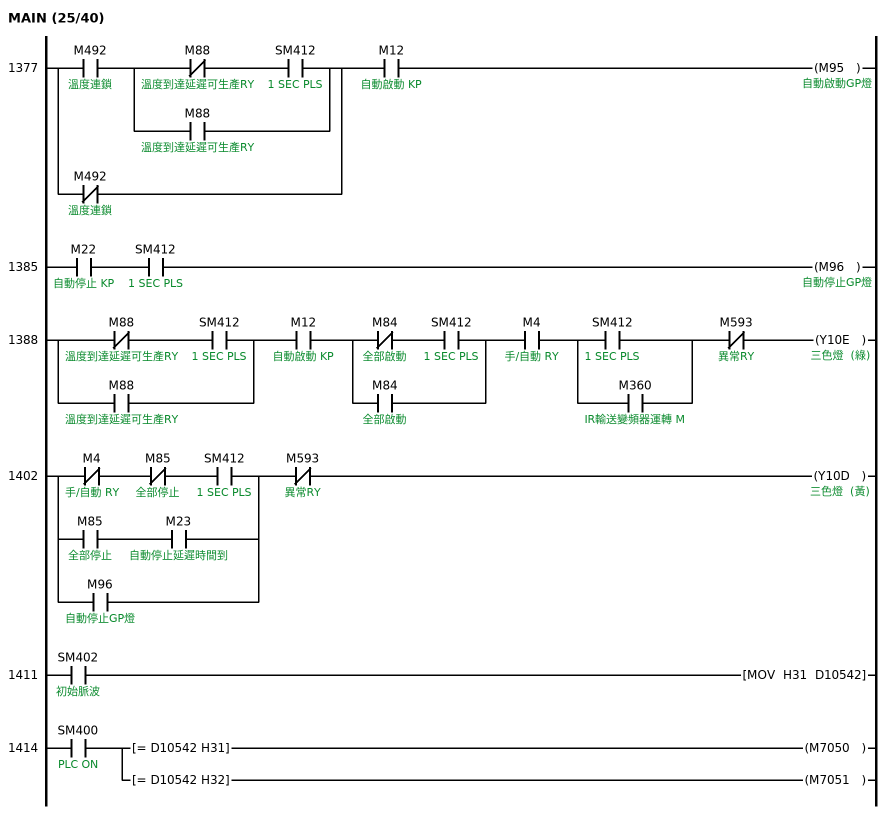
[picture p24: ladder of MAIN, rungs at steps 1377 to 1414]
1377  LD      M492  ; 溫度連鎖
      LDI     M88  ; 溫度到達延遲可生產RY
      AND     SM412  ; 1 SEC PLS
      OR      M88  ; 溫度到達延遲可生產RY
      ANB
      ORI     M492  ; 溫度連鎖
      AND     M12  ; 自動啟動 KP
      OUT     M95  ; 自動啟動GP燈
1385  LD      M22  ; 自動停止 KP
      AND     SM412  ; 1 SEC PLS
      OUT     M96  ; 自動停止GP燈
1388  LDI     M88  ; 溫度到達延遲可生產RY
      AND     SM412  ; 1 SEC PLS
      OR      M88  ; 溫度到達延遲可生產RY
      AND     M12  ; 自動啟動 KP
      LDI     M84  ; 全部啟動
      AND     SM412  ; 1 SEC PLS
      OR      M84  ; 全部啟動
      ANB
      AND     M4  ; 手/自動 RY
      LD      SM412  ; 1 SEC PLS
      OR      M360  ; IR輸送變頻器運轉 M
      ANB
      ANI     M593  ; 異常RY
      OUT     Y10E  ; 三色燈  (綠)
1402  LDI     M4  ; 手/自動 RY
      ANI     M85  ; 全部停止
      AND     SM412  ; 1 SEC PLS
      LD      M85  ; 全部停止
      AND     M23  ; 自動停止延遲時間到
      ORB
      OR      M96  ; 自動停止GP燈
      ANI     M593  ; 異常RY
      OUT     Y10D  ; 三色燈  (黃)
1411  LD      SM402  ; 初始脈波
      MOV     H31 D10542
1414  LD      SM400  ; PLC ON
      MPS
      AND=    D10542 H31
      OUT     M7050
      MPP
      AND=    D10542 H32
      OUT     M7051
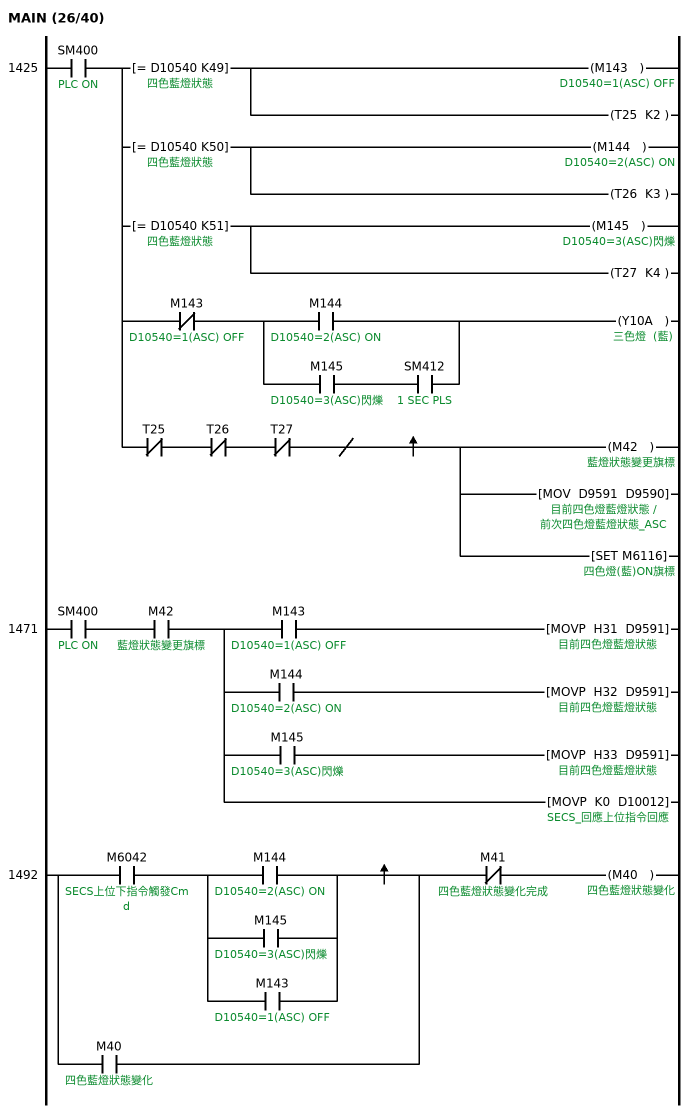
1425  LD      SM400  ; PLC ON
      MPS
      AND=    D10540 K49  ; 四色藍燈狀態
      OUT     M143  ; D10540=1(ASC) OFF
      OUT     T25 K2
      MRD
      AND=    D10540 K50  ; 四色藍燈狀態
      OUT     M144  ; D10540=2(ASC) ON
      OUT     T26 K3
      MRD
      AND=    D10540 K51  ; 四色藍燈狀態
      OUT     M145  ; D10540=3(ASC)閃爍
      OUT     T27 K4
      MRD
      ANI     M143  ; D10540=1(ASC) OFF
      LD      M144  ; D10540=2(ASC) ON
      LD      M145  ; D10540=3(ASC)閃爍
      AND     SM412  ; 1 SEC PLS
      ORB
      ANB
      OUT     Y10A  ; 三色燈  (藍)
      MPP
      ANI     T25
      ANI     T26
      ANI     T27
      INV
      MEP
      OUT     M42  ; 藍燈狀態變更旗標
      MOV     D9591 D9590  ; 目前四色燈藍燈狀態 / 前次四色燈藍燈狀態_ASC
      SET     M6116  ; 四色燈(藍)ON旗標
1471  LD      SM400  ; PLC ON
      AND     M42  ; 藍燈狀態變更旗標
      MPS
      AND     M143  ; D10540=1(ASC) OFF
      MOVP    H31 D9591
      MRD
      AND     M144  ; D10540=2(ASC) ON
      MOVP    H32 D9591
      MRD
      AND     M145  ; D10540=3(ASC)閃爍
      MOVP    H33 D9591
      MPP
      MOVP    K0 D10012  ; SECS_回應上位指令回應
1492  LD      M6042  ; SECS上位下指令觸發Cmd
      LD      M144  ; D10540=2(ASC) ON
      OR      M145  ; D10540=3(ASC)閃爍
      OR      M143  ; D10540=1(ASC) OFF
      ANB
      MEP
      OR      M40  ; 四色藍燈狀態變化
      ANI     M41  ; 四色藍燈狀態變化完成
      OUT     M40  ; 四色藍燈狀態變化
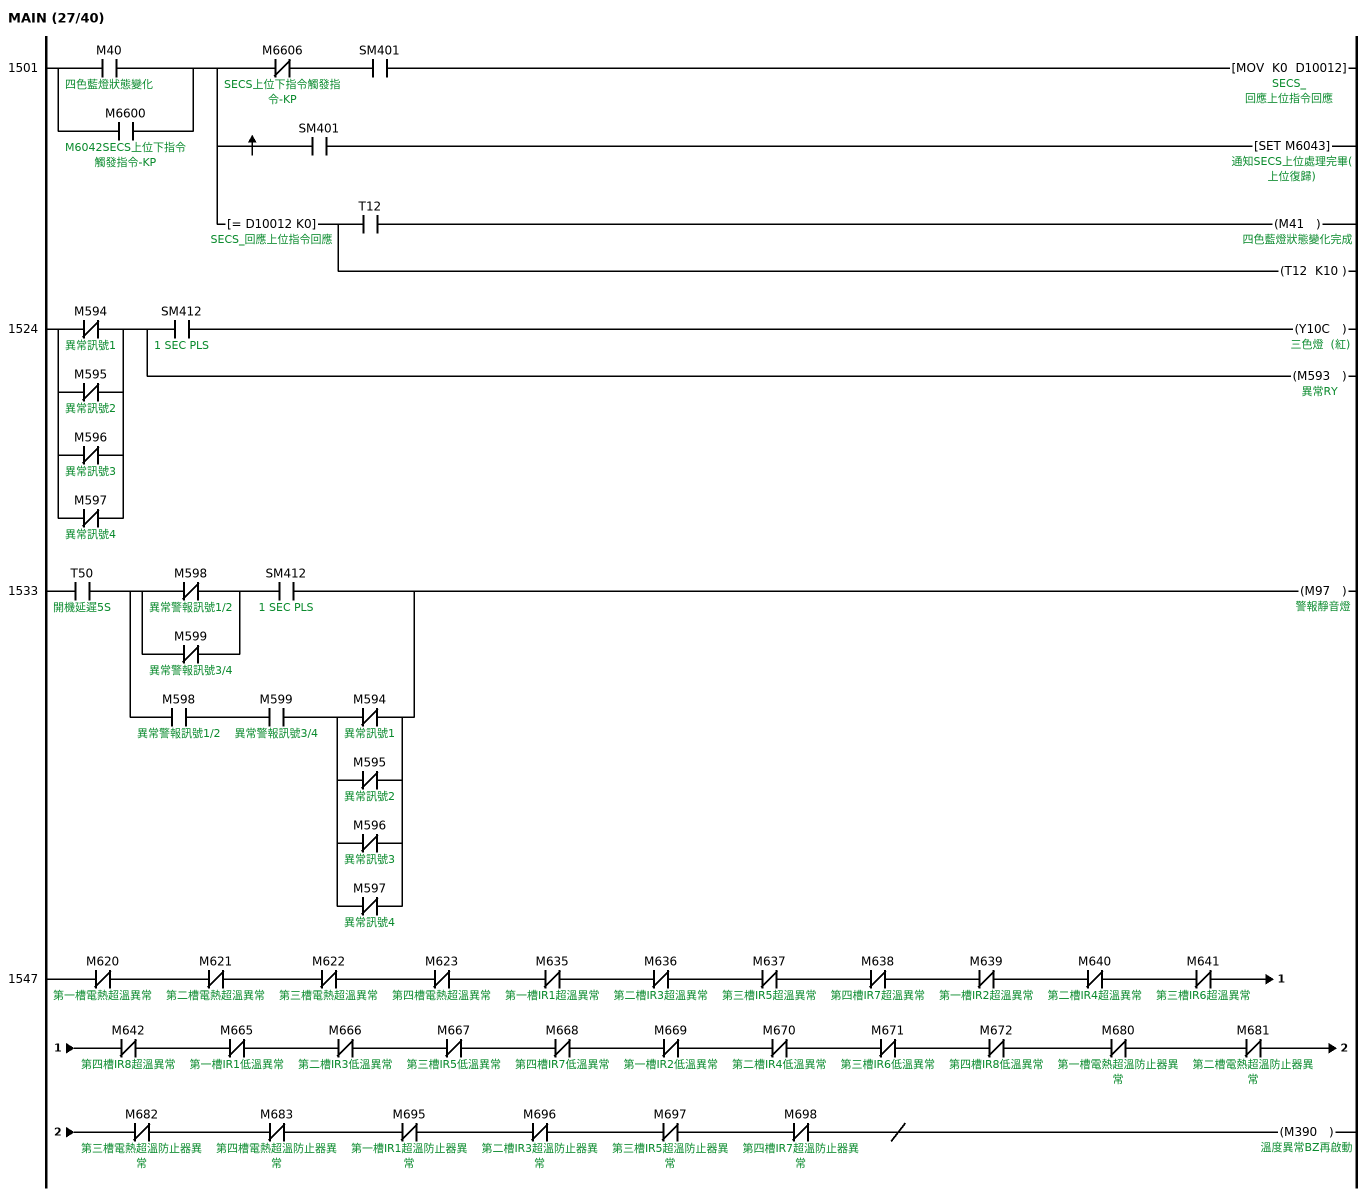
1501  LD      M40  ; 四色藍燈狀態變化
      OR      M6600  ; M6042SECS上位下指令觸發指令-KP
      MPS
      ANI     M6606  ; SECS上位下指令觸發指令-KP
      AND     SM401
      MOV     K0 D10012
      MRD
      MEP
      AND     SM401
      SET     M6043  ; 通知SECS上位處理完畢(上位復歸)
      MPP
      AND=    D10012 K0  ; SECS_回應上位指令回應
      MPS
      AND     T12
      OUT     M41  ; 四色藍燈狀態變化完成
      MPP
      OUT     T12 K10
1524  LDI     M594  ; 異常訊號1
      ORI     M595  ; 異常訊號2
      ORI     M596  ; 異常訊號3
      ORI     M597  ; 異常訊號4
      MPS
      AND     SM412  ; 1 SEC PLS
      OUT     Y10C  ; 三色燈  (紅)
      MPP
      OUT     M593  ; 異常RY
1533  LD      T50  ; 開機延遲5S
      LDI     M598  ; 異常警報訊號1/2
      ORI     M599  ; 異常警報訊號3/4
      AND     SM412  ; 1 SEC PLS
      LD      M598  ; 異常警報訊號1/2
      AND     M599  ; 異常警報訊號3/4
      LDI     M594  ; 異常訊號1
      ORI     M595  ; 異常訊號2
      ORI     M596  ; 異常訊號3
      ORI     M597  ; 異常訊號4
      ANB
      ORB
      ANB
      OUT     M97  ; 警報靜音燈
1547  LDI     M620  ; 第一槽電熱超溫異常
      ANI     M621  ; 第二槽電熱超溫異常
      ANI     M622  ; 第三槽電熱超溫異常
      ANI     M623  ; 第四槽電熱超溫異常
      ANI     M635  ; 第一槽IR1超溫異常
      ANI     M636  ; 第二槽IR3超溫異常
      ANI     M637  ; 第三槽IR5超溫異常
      ANI     M638  ; 第四槽IR7超溫異常
      ANI     M639  ; 第一槽IR2超溫異常
      ANI     M640  ; 第二槽IR4超溫異常
      ANI     M641  ; 第三槽IR6超溫異常
      ANI     M642  ; 第四槽IR8超溫異常
      ANI     M665  ; 第一槽IR1低溫異常
      ANI     M666  ; 第二槽IR3低溫異常
      ANI     M667  ; 第三槽IR5低溫異常
      ANI     M668  ; 第四槽IR7低溫異常
      ANI     M669  ; 第一槽IR2低溫異常
      ANI     M670  ; 第二槽IR4低溫異常
      ANI     M671  ; 第三槽IR6低溫異常
      ANI     M672  ; 第四槽IR8低溫異常
      ANI     M680  ; 第一槽電熱超溫防止器異常
      ANI     M681  ; 第二槽電熱超溫防止器異常
      ANI     M682  ; 第三槽電熱超溫防止器異常
      ANI     M683  ; 第四槽電熱超溫防止器異常
      ANI     M695  ; 第一槽IR1超溫防止器異常
      ANI     M696  ; 第二槽IR3超溫防止器異常
      ANI     M697  ; 第三槽IR5超溫防止器異常
      ANI     M698  ; 第四槽IR7超溫防止器異常
      INV
      OUT     M390  ; 溫度異常BZ再啟動
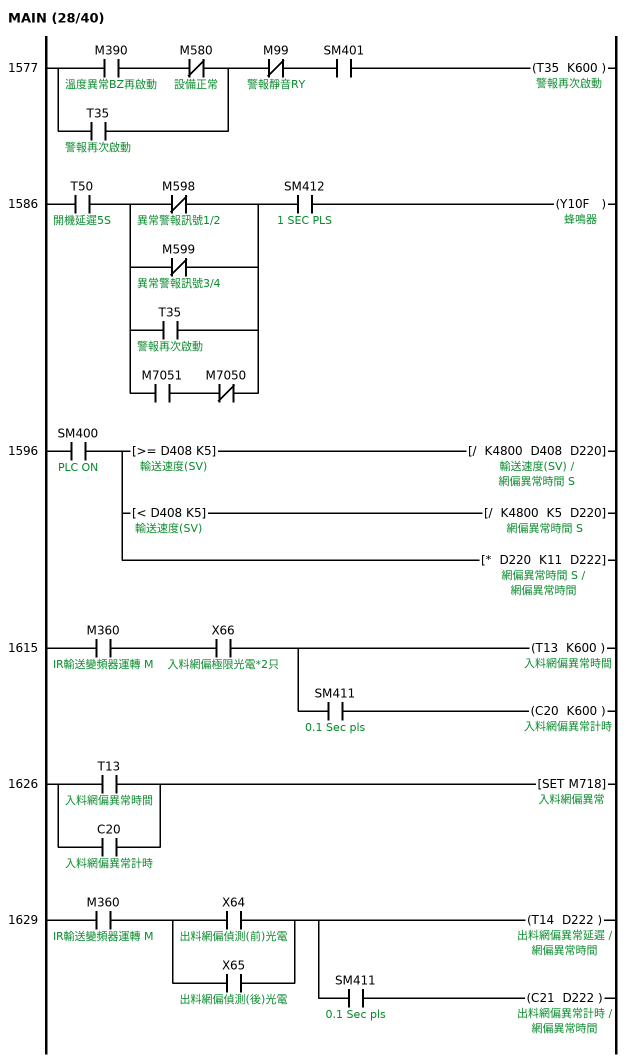
1577  LD      M390  ; 溫度異常BZ再啟動
      ANI     M580  ; 設備正常
      OR      T35  ; 警報再次啟動
      ANI     M99  ; 警報靜音RY
      AND     SM401
      OUT     T35 K600  ; 警報再次啟動
1586  LD      T50  ; 開機延遲5S
      LDI     M598  ; 異常警報訊號1/2
      ORI     M599  ; 異常警報訊號3/4
      OR      T35  ; 警報再次啟動
      LD      M7051
      ANI     M7050
      ORB
      ANB
      AND     SM412  ; 1 SEC PLS
      OUT     Y10F  ; 蜂鳴器
1596  LD      SM400  ; PLC ON
      MPS
      AND>=   D408 K5  ; 輸送速度(SV)
      /       K4800 D408 D220  ; 網偏異常時間 S
      MRD
      AND<    D408 K5  ; 輸送速度(SV)
      /       K4800 K5 D220
      MPP
      *       D220 K11 D222  ; 網偏異常時間
1615  LD      M360  ; IR輸送變頻器運轉 M
      AND     X66  ; 入料網偏極限光電*2只
      OUT     T13 K600  ; 入料網偏異常時間
      AND     SM411  ; 0.1 Sec pls
      OUT     C20 K600  ; 入料網偏異常計時
1626  LD      T13  ; 入料網偏異常時間
      OR      C20  ; 入料網偏異常計時
      SET     M718  ; 入料網偏異常
1629  LD      M360  ; IR輸送變頻器運轉 M
      LD      X64  ; 出料網偏偵測(前)光電
      OR      X65  ; 出料網偏偵測(後)光電
      ANB
      OUT     T14 D222  ; 出料網偏異常延遲 / 網偏異常時間
      AND     SM411  ; 0.1 Sec pls
      OUT     C21 D222  ; 出料網偏異常計時 / 網偏異常時間
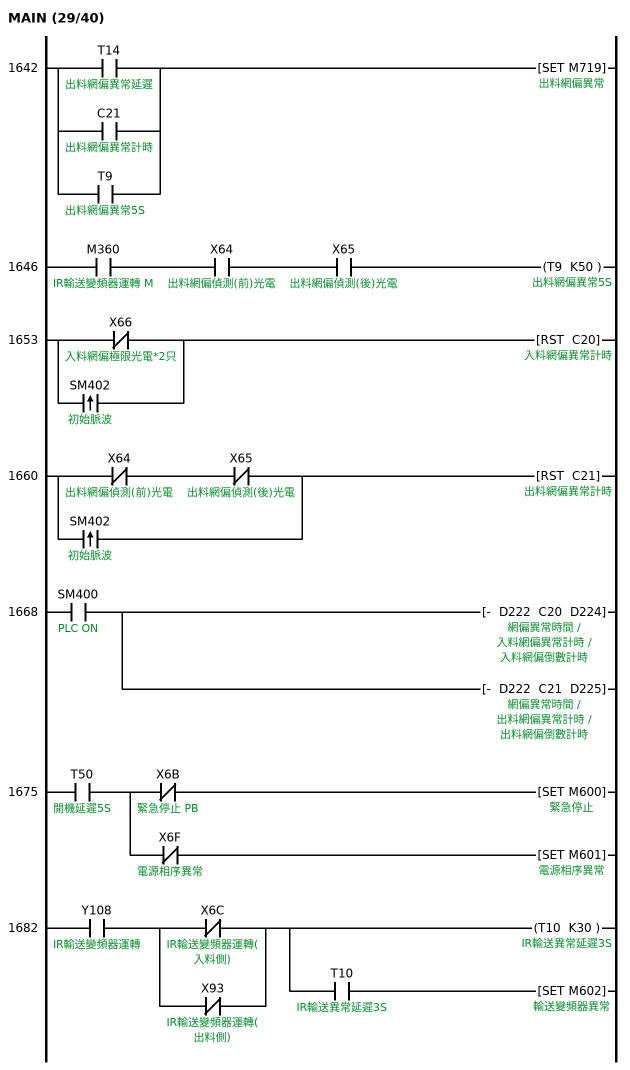
1642  LD      T14  ; 出料網偏異常延遲
      OR      C21  ; 出料網偏異常計時
      OR      T9  ; 出料網偏異常5S
      SET     M719  ; 出料網偏異常
1646  LD      M360  ; IR輸送變頻器運轉 M
      AND     X64  ; 出料網偏偵測(前)光電
      AND     X65  ; 出料網偏偵測(後)光電
      OUT     T9 K50  ; 出料網偏異常5S
1653  LDI     X66  ; 入料網偏極限光電*2只
      ORP     SM402  ; 初始脈波
      RST     C20  ; 入料網偏異常計時
1660  LDI     X64  ; 出料網偏偵測(前)光電
      ANI     X65  ; 出料網偏偵測(後)光電
      ORP     SM402  ; 初始脈波
      RST     C21  ; 出料網偏異常計時
1668  LD      SM400  ; PLC ON
      -       D222 C20 D224  ; 入料網偏倒數計時
      -       D222 C21 D225  ; 出料網偏倒數計時
1675  LD      T50  ; 開機延遲5S
      MPS
      ANI     X6B  ; 緊急停止 PB
      SET     M600  ; 緊急停止
      MPP
      ANI     X6F  ; 電源相序異常
      SET     M601  ; 電源相序異常
1682  LD      Y108  ; IR輸送變頻器運轉
      LDI     X6C  ; IR輸送變頻器運轉(入料側)
      ORI     X93  ; IR輸送變頻器運轉(出料側)
      ANB
      OUT     T10 K30  ; IR輸送異常延遲3S
      AND     T10  ; IR輸送異常延遲3S
      SET     M602  ; 輸送變頻器異常
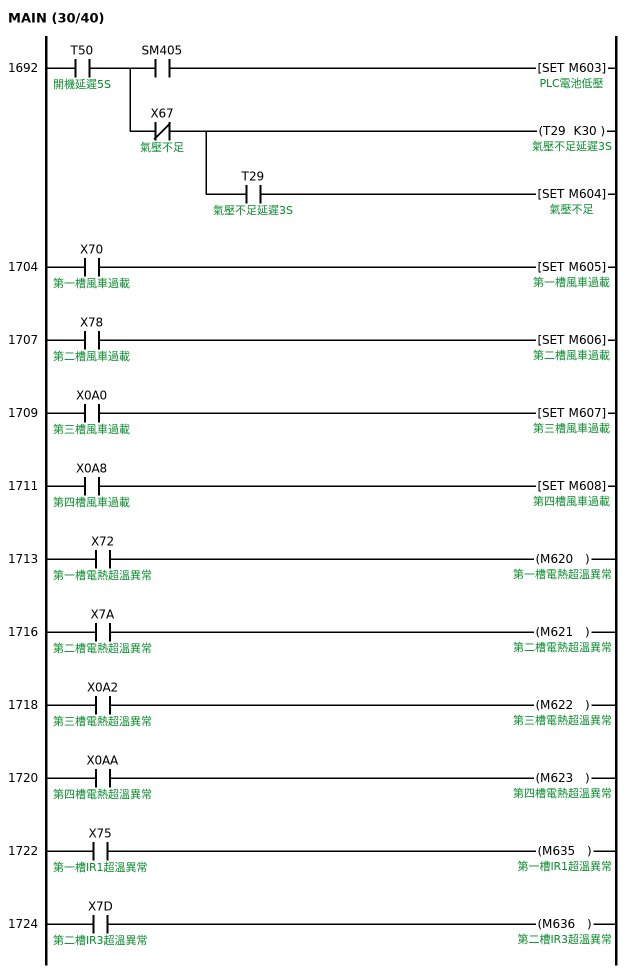
1692  LD      T50  ; 開機延遲5S
      MPS
      AND     SM405
      SET     M603  ; PLC電池低壓
      MPP
      ANI     X67  ; 氣壓不足
      OUT     T29 K30  ; 氣壓不足延遲3S
      AND     T29  ; 氣壓不足延遲3S
      SET     M604  ; 氣壓不足
1704  LD      X70  ; 第一槽風車過載
      SET     M605  ; 第一槽風車過載
        [note] 
1707  LD      X78  ; 第二槽風車過載
      SET     M606  ; 第二槽風車過載
1709  LD      X0A0  ; 第三槽風車過載
      SET     M607  ; 第三槽風車過載
1711  LD      X0A8  ; 第四槽風車過載
      SET     M608  ; 第四槽風車過載
1713  LD      X72  ; 第一槽電熱超溫異常
      OUT     M620  ; 第一槽電熱超溫異常
        [note] 
1716  LD      X7A  ; 第二槽電熱超溫異常
      OUT     M621  ; 第二槽電熱超溫異常
1718  LD      X0A2  ; 第三槽電熱超溫異常
      OUT     M622  ; 第三槽電熱超溫異常
1720  LD      X0AA  ; 第四槽電熱超溫異常
      OUT     M623  ; 第四槽電熱超溫異常
1722  LD      X75  ; 第一槽IR1超溫異常
      OUT     M635  ; 第一槽IR1超溫異常
1724  LD      X7D  ; 第二槽IR3超溫異常
      OUT     M636  ; 第二槽IR3超溫異常
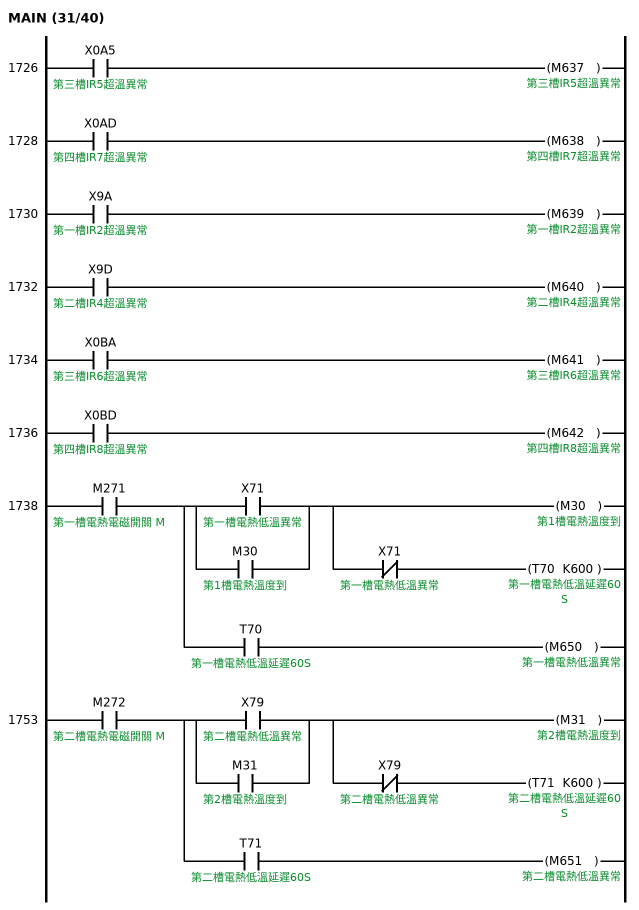
1726  LD      X0A5  ; 第三槽IR5超溫異常
      OUT     M637  ; 第三槽IR5超溫異常
1728  LD      X0AD  ; 第四槽IR7超溫異常
      OUT     M638  ; 第四槽IR7超溫異常
1730  LD      X9A  ; 第一槽IR2超溫異常
      OUT     M639  ; 第一槽IR2超溫異常
1732  LD      X9D  ; 第二槽IR4超溫異常
      OUT     M640  ; 第二槽IR4超溫異常
1734  LD      X0BA  ; 第三槽IR6超溫異常
      OUT     M641  ; 第三槽IR6超溫異常
1736  LD      X0BD  ; 第四槽IR8超溫異常
      OUT     M642  ; 第四槽IR8超溫異常
1738  LD      M271  ; 第一槽電熱電磁開關 M
      MPS
      LD      X71  ; 第一槽電熱低溫異常
      OR      M30  ; 第1槽電熱溫度到
      ANB
      OUT     M30  ; 第1槽電熱溫度到
        [note] 
      ANI     X71  ; 第一槽電熱低溫異常
      OUT     T70 K600  ; 第一槽電熱低溫延遲60S
      MPP
      AND     T70  ; 第一槽電熱低溫延遲60S
      OUT     M650  ; 第一槽電熱低溫異常
1753  LD      M272  ; 第二槽電熱電磁開關 M
      MPS
      LD      X79  ; 第二槽電熱低溫異常
      OR      M31  ; 第2槽電熱溫度到
      ANB
      OUT     M31  ; 第2槽電熱溫度到
      ANI     X79  ; 第二槽電熱低溫異常
      OUT     T71 K600  ; 第二槽電熱低溫延遲60S
      MPP
      AND     T71  ; 第二槽電熱低溫延遲60S
      OUT     M651  ; 第二槽電熱低溫異常
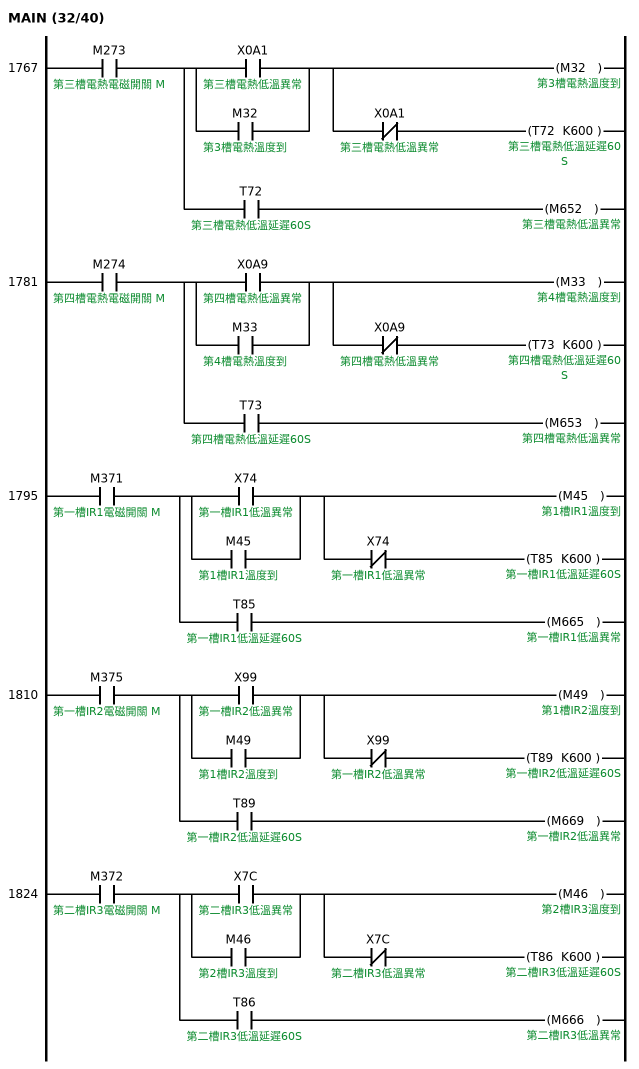
1767  LD      M273  ; 第三槽電熱電磁開關 M
      MPS
      LD      X0A1  ; 第三槽電熱低溫異常
      OR      M32  ; 第3槽電熱溫度到
      ANB
      OUT     M32  ; 第3槽電熱溫度到
      ANI     X0A1  ; 第三槽電熱低溫異常
      OUT     T72 K600  ; 第三槽電熱低溫延遲60S
      MPP
      AND     T72  ; 第三槽電熱低溫延遲60S
      OUT     M652  ; 第三槽電熱低溫異常
1781  LD      M274  ; 第四槽電熱電磁開關 M
      MPS
      LD      X0A9  ; 第四槽電熱低溫異常
      OR      M33  ; 第4槽電熱溫度到
      ANB
      OUT     M33  ; 第4槽電熱溫度到
      ANI     X0A9  ; 第四槽電熱低溫異常
      OUT     T73 K600  ; 第四槽電熱低溫延遲60S
      MPP
      AND     T73  ; 第四槽電熱低溫延遲60S
      OUT     M653  ; 第四槽電熱低溫異常
1795  LD      M371  ; 第一槽IR1電磁開關 M
      MPS
      LD      X74  ; 第一槽IR1低溫異常
      OR      M45  ; 第1槽IR1溫度到
      ANB
      OUT     M45  ; 第1槽IR1溫度到
        [note] 
      ANI     X74  ; 第一槽IR1低溫異常
      OUT     T85 K600  ; 第一槽IR1低溫延遲60S
      MPP
      AND     T85  ; 第一槽IR1低溫延遲60S
      OUT     M665  ; 第一槽IR1低溫異常
1810  LD      M375  ; 第一槽IR2電磁開關 M
      MPS
      LD      X99  ; 第一槽IR2低溫異常
      OR      M49  ; 第1槽IR2溫度到
      ANB
      OUT     M49  ; 第1槽IR2溫度到
      ANI     X99  ; 第一槽IR2低溫異常
      OUT     T89 K600  ; 第一槽IR2低溫延遲60S
      MPP
      AND     T89  ; 第一槽IR2低溫延遲60S
      OUT     M669  ; 第一槽IR2低溫異常
1824  LD      M372  ; 第二槽IR3電磁開關 M
      MPS
      LD      X7C  ; 第二槽IR3低溫異常
      OR      M46  ; 第2槽IR3溫度到
      ANB
      OUT     M46  ; 第2槽IR3溫度到
      ANI     X7C  ; 第二槽IR3低溫異常
      OUT     T86 K600  ; 第二槽IR3低溫延遲60S
      MPP
      AND     T86  ; 第二槽IR3低溫延遲60S
      OUT     M666  ; 第二槽IR3低溫異常
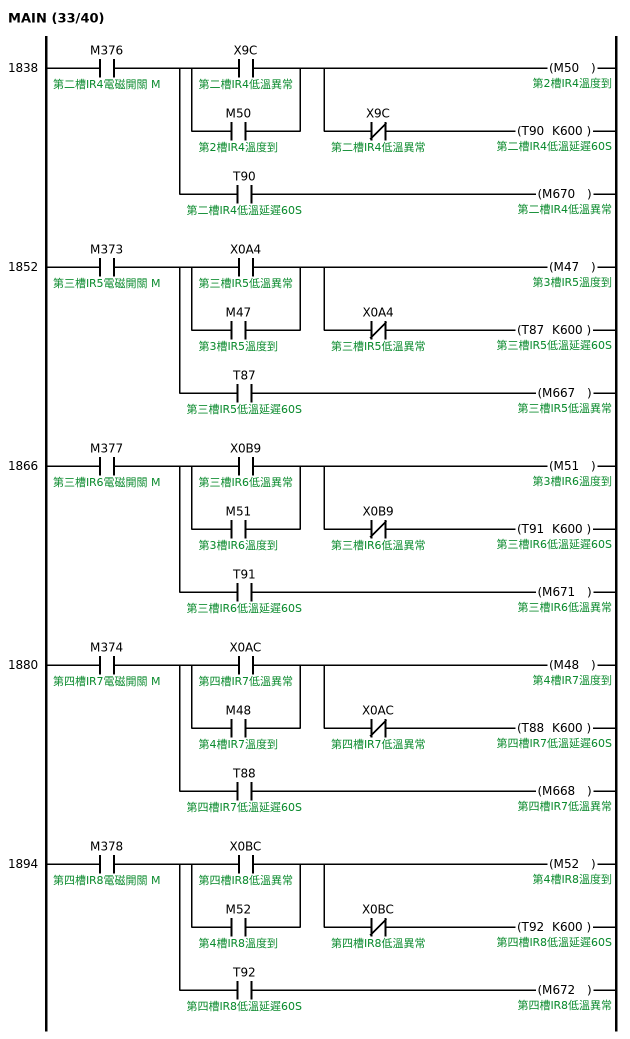
1838  LD      M376  ; 第二槽IR4電磁開關 M
      MPS
      LD      X9C  ; 第二槽IR4低溫異常
      OR      M50  ; 第2槽IR4溫度到
      ANB
      OUT     M50  ; 第2槽IR4溫度到
      ANI     X9C  ; 第二槽IR4低溫異常
      OUT     T90 K600  ; 第二槽IR4低溫延遲60S
      MPP
      AND     T90  ; 第二槽IR4低溫延遲60S
      OUT     M670  ; 第二槽IR4低溫異常
1852  LD      M373  ; 第三槽IR5電磁開關 M
      MPS
      LD      X0A4  ; 第三槽IR5低溫異常
      OR      M47  ; 第3槽IR5溫度到
      ANB
      OUT     M47  ; 第3槽IR5溫度到
      ANI     X0A4  ; 第三槽IR5低溫異常
      OUT     T87 K600  ; 第三槽IR5低溫延遲60S
      MPP
      AND     T87  ; 第三槽IR5低溫延遲60S
      OUT     M667  ; 第三槽IR5低溫異常
1866  LD      M377  ; 第三槽IR6電磁開關 M
      MPS
      LD      X0B9  ; 第三槽IR6低溫異常
      OR      M51  ; 第3槽IR6溫度到
      ANB
      OUT     M51  ; 第3槽IR6溫度到
      ANI     X0B9  ; 第三槽IR6低溫異常
      OUT     T91 K600  ; 第三槽IR6低溫延遲60S
      MPP
      AND     T91  ; 第三槽IR6低溫延遲60S
      OUT     M671  ; 第三槽IR6低溫異常
1880  LD      M374  ; 第四槽IR7電磁開關 M
      MPS
      LD      X0AC  ; 第四槽IR7低溫異常
      OR      M48  ; 第4槽IR7溫度到
      ANB
      OUT     M48  ; 第4槽IR7溫度到
      ANI     X0AC  ; 第四槽IR7低溫異常
      OUT     T88 K600  ; 第四槽IR7低溫延遲60S
      MPP
      AND     T88  ; 第四槽IR7低溫延遲60S
      OUT     M668  ; 第四槽IR7低溫異常
1894  LD      M378  ; 第四槽IR8電磁開關 M
      MPS
      LD      X0BC  ; 第四槽IR8低溫異常
      OR      M52  ; 第4槽IR8溫度到
      ANB
      OUT     M52  ; 第4槽IR8溫度到
      ANI     X0BC  ; 第四槽IR8低溫異常
      OUT     T92 K600  ; 第四槽IR8低溫延遲60S
      MPP
      AND     T92  ; 第四槽IR8低溫延遲60S
      OUT     M672  ; 第四槽IR8低溫異常
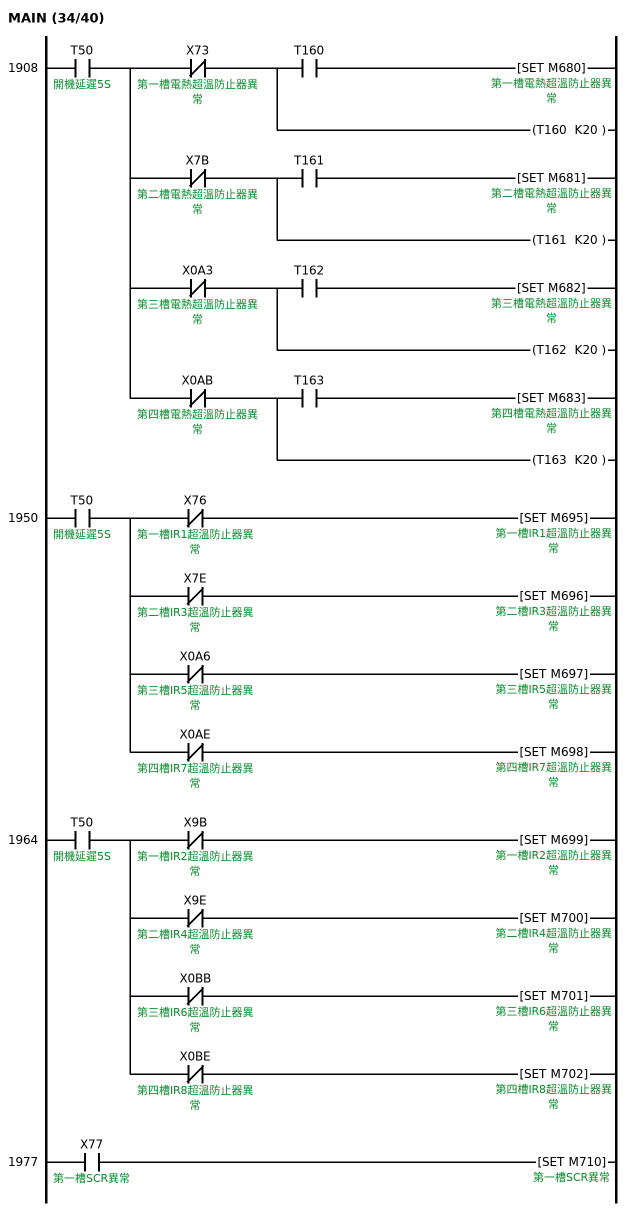
1908  LD      T50  ; 開機延遲5S
      MPS
      ANI     X73  ; 第一槽電熱超溫防止器異常
      MPS
      AND     T160
      SET     M680  ; 第一槽電熱超溫防止器異常
        [note] 
      MPP
      OUT     T160 K20
      MRD
      ANI     X7B  ; 第二槽電熱超溫防止器異常
      MPS
      AND     T161
      SET     M681  ; 第二槽電熱超溫防止器異常
      MPP
      OUT     T161 K20
      MRD
      ANI     X0A3  ; 第三槽電熱超溫防止器異常
      MPS
      AND     T162
      SET     M682  ; 第三槽電熱超溫防止器異常
      MPP
      OUT     T162 K20
      MPP
      ANI     X0AB  ; 第四槽電熱超溫防止器異常
      MPS
      AND     T163
      SET     M683  ; 第四槽電熱超溫防止器異常
      MPP
      OUT     T163 K20
1950  LD      T50  ; 開機延遲5S
      MPS
      ANI     X76  ; 第一槽IR1超溫防止器異常
      SET     M695  ; 第一槽IR1超溫防止器異常
        [note] 
      MRD
      ANI     X7E  ; 第二槽IR3超溫防止器異常
      SET     M696  ; 第二槽IR3超溫防止器異常
      MRD
      ANI     X0A6  ; 第三槽IR5超溫防止器異常
      SET     M697  ; 第三槽IR5超溫防止器異常
      MPP
      ANI     X0AE  ; 第四槽IR7超溫防止器異常
      SET     M698  ; 第四槽IR7超溫防止器異常
1964  LD      T50  ; 開機延遲5S
      MPS
      ANI     X9B  ; 第一槽IR2超溫防止器異常
      SET     M699  ; 第一槽IR2超溫防止器異常
      MRD
      ANI     X9E  ; 第二槽IR4超溫防止器異常
      SET     M700  ; 第二槽IR4超溫防止器異常
      MRD
      ANI     X0BB  ; 第三槽IR6超溫防止器異常
      SET     M701  ; 第三槽IR6超溫防止器異常
      MPP
      ANI     X0BE  ; 第四槽IR8超溫防止器異常
      SET     M702  ; 第四槽IR8超溫防止器異常
1977  LD      X77  ; 第一槽SCR異常
      SET     M710  ; 第一槽SCR異常
        [note] 
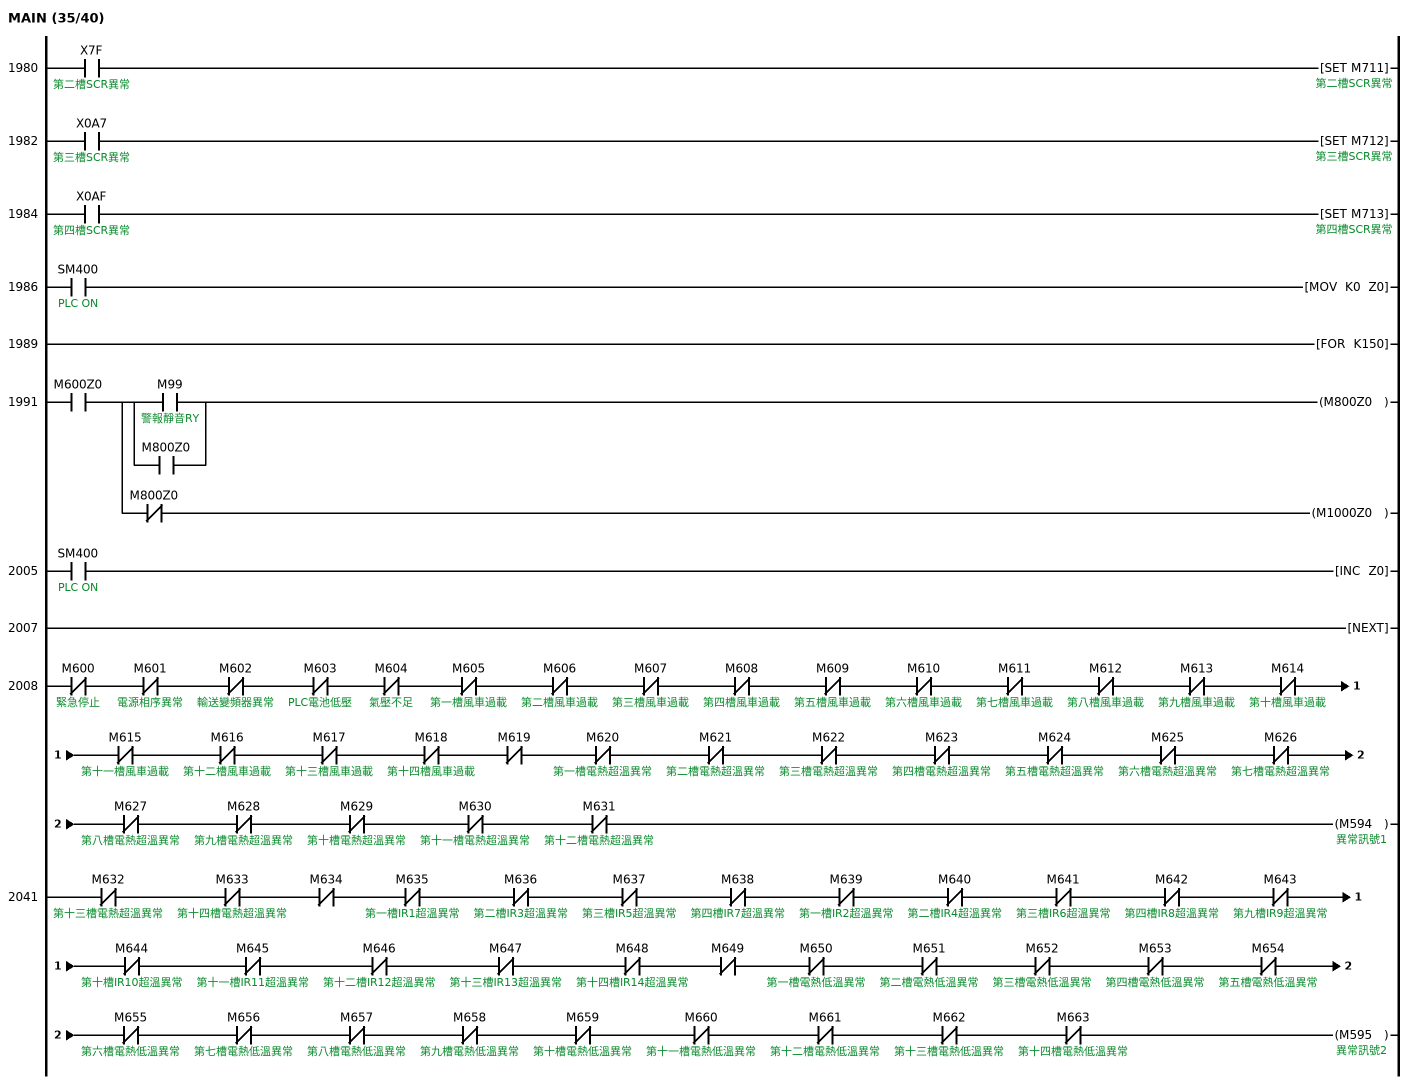
1980  LD      X7F  ; 第二槽SCR異常
      SET     M711  ; 第二槽SCR異常
1982  LD      X0A7  ; 第三槽SCR異常
      SET     M712  ; 第三槽SCR異常
1984  LD      X0AF  ; 第四槽SCR異常
      SET     M713  ; 第四槽SCR異常
1986  LD      SM400  ; PLC ON
      MOV     K0 Z0
1989  FOR     K150
1991  LD      M600Z0
      MPS
      LD      M99  ; 警報靜音RY
      OR      M800Z0
      ANB
      OUT     M800Z0
      MPP
      ANI     M800Z0
      OUT     M1000Z0
2005  LD      SM400  ; PLC ON
      INC     Z0
2007  NEXT
2008  LDI     M600  ; 緊急停止
      ANI     M601  ; 電源相序異常
      ANI     M602  ; 輸送變頻器異常
      ANI     M603  ; PLC電池低壓
      ANI     M604  ; 氣壓不足
      ANI     M605  ; 第一槽風車過載
      ANI     M606  ; 第二槽風車過載
      ANI     M607  ; 第三槽風車過載
      ANI     M608  ; 第四槽風車過載
      ANI     M609  ; 第五槽風車過載
      ANI     M610  ; 第六槽風車過載
      ANI     M611  ; 第七槽風車過載
      ANI     M612  ; 第八槽風車過載
      ANI     M613  ; 第九槽風車過載
      ANI     M614  ; 第十槽風車過載
      ANI     M615  ; 第十一槽風車過載
      ANI     M616  ; 第十二槽風車過載
      ANI     M617  ; 第十三槽風車過載
      ANI     M618  ; 第十四槽風車過載
      ANI     M619
      ANI     M620  ; 第一槽電熱超溫異常
      ANI     M621  ; 第二槽電熱超溫異常
      ANI     M622  ; 第三槽電熱超溫異常
      ANI     M623  ; 第四槽電熱超溫異常
      ANI     M624  ; 第五槽電熱超溫異常
      ANI     M625  ; 第六槽電熱超溫異常
      ANI     M626  ; 第七槽電熱超溫異常
      ANI     M627  ; 第八槽電熱超溫異常
      ANI     M628  ; 第九槽電熱超溫異常
      ANI     M629  ; 第十槽電熱超溫異常
      ANI     M630  ; 第十一槽電熱超溫異常
      ANI     M631  ; 第十二槽電熱超溫異常
      OUT     M594  ; 異常訊號1
2041  LDI     M632  ; 第十三槽電熱超溫異常
      ANI     M633  ; 第十四槽電熱超溫異常
      ANI     M634
      ANI     M635  ; 第一槽IR1超溫異常
      ANI     M636  ; 第二槽IR3超溫異常
      ANI     M637  ; 第三槽IR5超溫異常
      ANI     M638  ; 第四槽IR7超溫異常
      ANI     M639  ; 第一槽IR2超溫異常
      ANI     M640  ; 第二槽IR4超溫異常
      ANI     M641  ; 第三槽IR6超溫異常
      ANI     M642  ; 第四槽IR8超溫異常
      ANI     M643  ; 第九槽IR9超溫異常
      ANI     M644  ; 第十槽IR10超溫異常
      ANI     M645  ; 第十一槽IR11超溫異常
      ANI     M646  ; 第十二槽IR12超溫異常
      ANI     M647  ; 第十三槽IR13超溫異常
      ANI     M648  ; 第十四槽IR14超溫異常
      ANI     M649
      ANI     M650  ; 第一槽電熱低溫異常
      ANI     M651  ; 第二槽電熱低溫異常
      ANI     M652  ; 第三槽電熱低溫異常
      ANI     M653  ; 第四槽電熱低溫異常
      ANI     M654  ; 第五槽電熱低溫異常
      ANI     M655  ; 第六槽電熱低溫異常
      ANI     M656  ; 第七槽電熱低溫異常
      ANI     M657  ; 第八槽電熱低溫異常
      ANI     M658  ; 第九槽電熱低溫異常
      ANI     M659  ; 第十槽電熱低溫異常
      ANI     M660  ; 第十一槽電熱低溫異常
      ANI     M661  ; 第十二槽電熱低溫異常
      ANI     M662  ; 第十三槽電熱低溫異常
      ANI     M663  ; 第十四槽電熱低溫異常
      OUT     M595  ; 異常訊號2
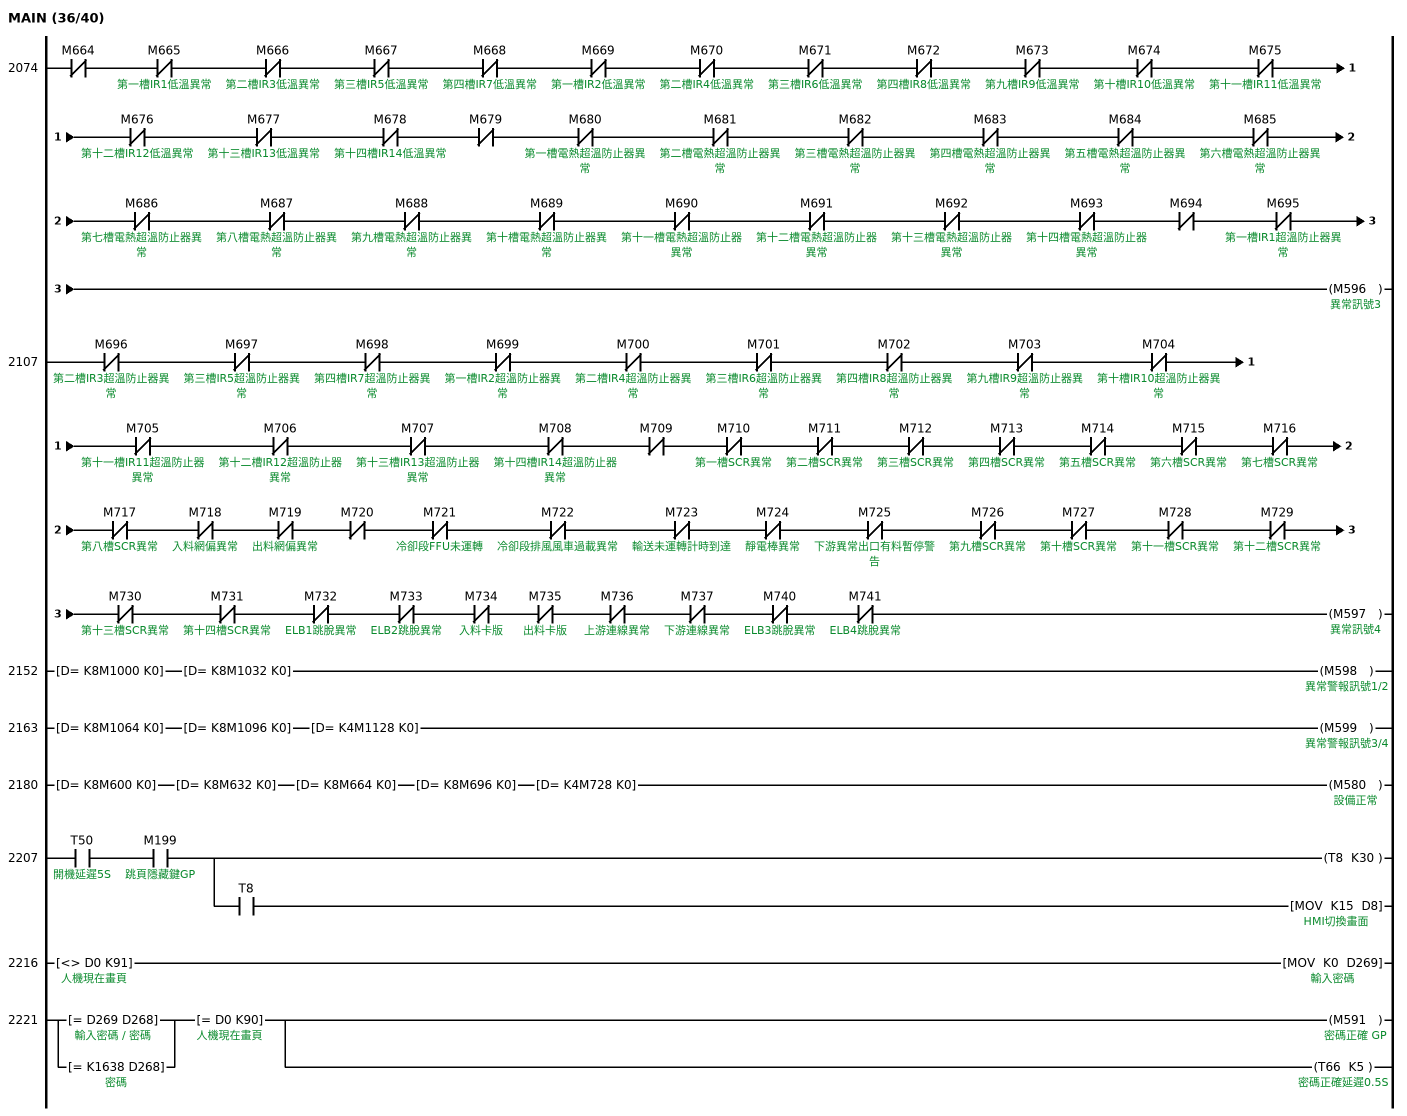
2074  LDI     M664
      ANI     M665  ; 第一槽IR1低溫異常
      ANI     M666  ; 第二槽IR3低溫異常
      ANI     M667  ; 第三槽IR5低溫異常
      ANI     M668  ; 第四槽IR7低溫異常
      ANI     M669  ; 第一槽IR2低溫異常
      ANI     M670  ; 第二槽IR4低溫異常
      ANI     M671  ; 第三槽IR6低溫異常
      ANI     M672  ; 第四槽IR8低溫異常
      ANI     M673  ; 第九槽IR9低溫異常
      ANI     M674  ; 第十槽IR10低溫異常
      ANI     M675  ; 第十一槽IR11低溫異常
      ANI     M676  ; 第十二槽IR12低溫異常
      ANI     M677  ; 第十三槽IR13低溫異常
      ANI     M678  ; 第十四槽IR14低溫異常
      ANI     M679
      ANI     M680  ; 第一槽電熱超溫防止器異常
      ANI     M681  ; 第二槽電熱超溫防止器異常
      ANI     M682  ; 第三槽電熱超溫防止器異常
      ANI     M683  ; 第四槽電熱超溫防止器異常
      ANI     M684  ; 第五槽電熱超溫防止器異常
      ANI     M685  ; 第六槽電熱超溫防止器異常
      ANI     M686  ; 第七槽電熱超溫防止器異常
      ANI     M687  ; 第八槽電熱超溫防止器異常
      ANI     M688  ; 第九槽電熱超溫防止器異常
      ANI     M689  ; 第十槽電熱超溫防止器異常
      ANI     M690  ; 第十一槽電熱超溫防止器異常
      ANI     M691  ; 第十二槽電熱超溫防止器異常
      ANI     M692  ; 第十三槽電熱超溫防止器異常
      ANI     M693  ; 第十四槽電熱超溫防止器異常
      ANI     M694
      ANI     M695  ; 第一槽IR1超溫防止器異常
      OUT     M596  ; 異常訊號3
2107  LDI     M696  ; 第二槽IR3超溫防止器異常
      ANI     M697  ; 第三槽IR5超溫防止器異常
      ANI     M698  ; 第四槽IR7超溫防止器異常
      ANI     M699  ; 第一槽IR2超溫防止器異常
      ANI     M700  ; 第二槽IR4超溫防止器異常
      ANI     M701  ; 第三槽IR6超溫防止器異常
      ANI     M702  ; 第四槽IR8超溫防止器異常
      ANI     M703  ; 第九槽IR9超溫防止器異常
      ANI     M704  ; 第十槽IR10超溫防止器異常
      ANI     M705  ; 第十一槽IR11超溫防止器異常
      ANI     M706  ; 第十二槽IR12超溫防止器異常
      ANI     M707  ; 第十三槽IR13超溫防止器異常
      ANI     M708  ; 第十四槽IR14超溫防止器異常
      ANI     M709
      ANI     M710  ; 第一槽SCR異常
      ANI     M711  ; 第二槽SCR異常
      ANI     M712  ; 第三槽SCR異常
      ANI     M713  ; 第四槽SCR異常
      ANI     M714  ; 第五槽SCR異常
      ANI     M715  ; 第六槽SCR異常
      ANI     M716  ; 第七槽SCR異常
      ANI     M717  ; 第八槽SCR異常
      ANI     M718  ; 入料網偏異常
      ANI     M719  ; 出料網偏異常
      ANI     M720
      ANI     M721  ; 冷卻段FFU未運轉
      ANI     M722  ; 冷卻段排風風車過載異常
      ANI     M723  ; 輸送未運轉計時到達
      ANI     M724  ; 靜電棒異常
      ANI     M725  ; 下游異常出口有料暫停警告
      ANI     M726  ; 第九槽SCR異常
      ANI     M727  ; 第十槽SCR異常
      ANI     M728  ; 第十一槽SCR異常
      ANI     M729  ; 第十二槽SCR異常
      ANI     M730  ; 第十三槽SCR異常
      ANI     M731  ; 第十四槽SCR異常
      ANI     M732  ; ELB1跳脫異常
      ANI     M733  ; ELB2跳脫異常
      ANI     M734  ; 入料卡版
      ANI     M735  ; 出料卡版
      ANI     M736  ; 上游連線異常
      ANI     M737  ; 下游連線異常
      ANI     M740  ; ELB3跳脫異常
      ANI     M741  ; ELB4跳脫異常
      OUT     M597  ; 異常訊號4
2152  LDD=    K8M1000 K0  ; 緊急停止迴圈資料
      ANDD=   K8M1032 K0  ; 迴圈資料
      OUT     M598  ; 異常警報訊號1/2
2163  LDD=    K8M1064 K0  ; 迴圈資料
      ANDD=   K8M1096 K0  ; 迴圈資料
      ANDD=   K4M1128 K0
      OUT     M599  ; 異常警報訊號3/4
2180  LDD=    K8M600 K0  ; 緊急停止
      ANDD=   K8M632 K0  ; 第十三槽電熱超溫異常
      ANDD=   K8M664 K0
      ANDD=   K8M696 K0  ; 第二槽IR3超溫防止器異常
      ANDD=   K4M728 K0  ; 第十一槽SCR異常
      OUT     M580  ; 設備正常
2207  LD      T50  ; 開機延遲5S
      AND     M199  ; 跳頁隱藏鍵GP
      OUT     T8 K30
      AND     T8
      MOV     K15 D8  ; HMI切換畫面
2216  LD<>    D0 K91  ; 人機現在畫頁
      MOV     K0 D269  ; 輸入密碼
2221  LD=     D269 D268  ; 輸入密碼 / 密碼
      OR=     K1638 D268  ; 密碼
      AND=    D0 K90  ; 人機現在畫頁
      OUT     M591  ; 密碼正確 GP
      OUT     T66 K5  ; 密碼正確延遲0.5S
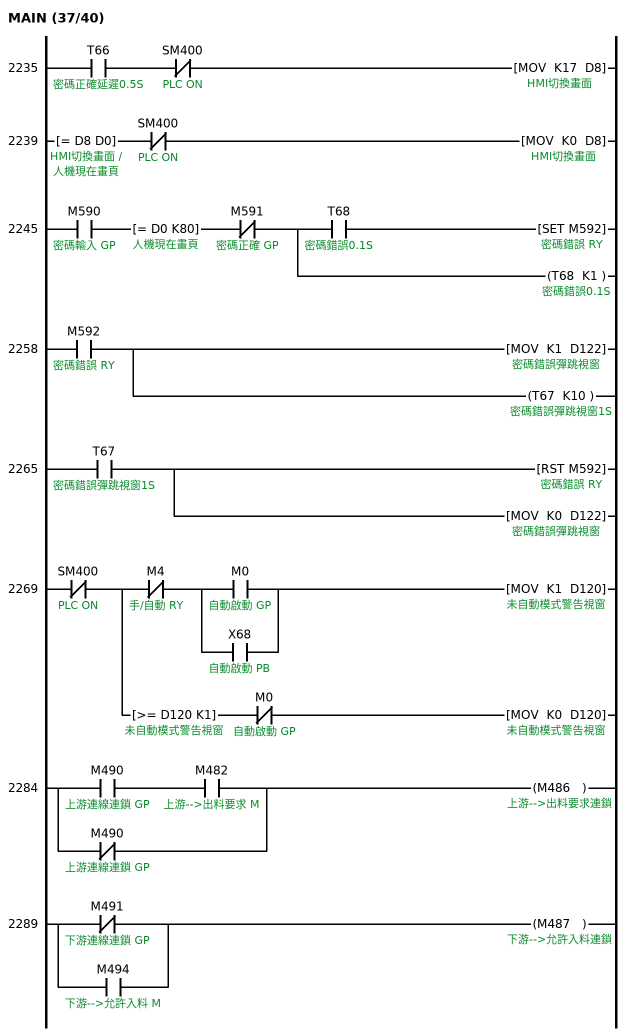
2235  LD      T66  ; 密碼正確延遲0.5S
      ANI     SM400  ; PLC ON
      MOV     K17 D8
2239  LD=     D8 D0  ; HMI切換畫面 / 人機現在畫頁
      ANI     SM400  ; PLC ON
      MOV     K0 D8
2245  LD      M590  ; 密碼輸入 GP
      AND=    D0 K80  ; 人機現在畫頁
      ANI     M591  ; 密碼正確 GP
      MPS
      AND     T68  ; 密碼錯誤0.1S
      SET     M592  ; 密碼錯誤 RY
      MPP
      OUT     T68 K1  ; 密碼錯誤0.1S
2258  LD      M592  ; 密碼錯誤 RY
      MOV     K1 D122  ; 密碼錯誤彈跳視窗
      OUT     T67 K10  ; 密碼錯誤彈跳視窗1S
2265  LD      T67  ; 密碼錯誤彈跳視窗1S
      RST     M592  ; 密碼錯誤 RY
      MOV     K0 D122
2269  LDI     SM400  ; PLC ON
      MPS
      ANI     M4  ; 手/自動 RY
      LD      M0  ; 自動啟動 GP
      OR      X68  ; 自動啟動 PB
      ANB
      MOV     K1 D120  ; 未自動模式警告視窗
      MPP
      AND>=   D120 K1  ; 未自動模式警告視窗
      ANI     M0  ; 自動啟動 GP
      MOV     K0 D120
2284  LD      M490  ; 上游連線連鎖 GP
      AND     M482  ; 上游-->出料要求 M
      ORI     M490  ; 上游連線連鎖 GP
      OUT     M486  ; 上游-->出料要求連鎖
        [note] 
2289  LDI     M491  ; 下游連線連鎖 GP
      OR      M494  ; 下游-->允許入料 M
      OUT     M487  ; 下游-->允許入料連鎖
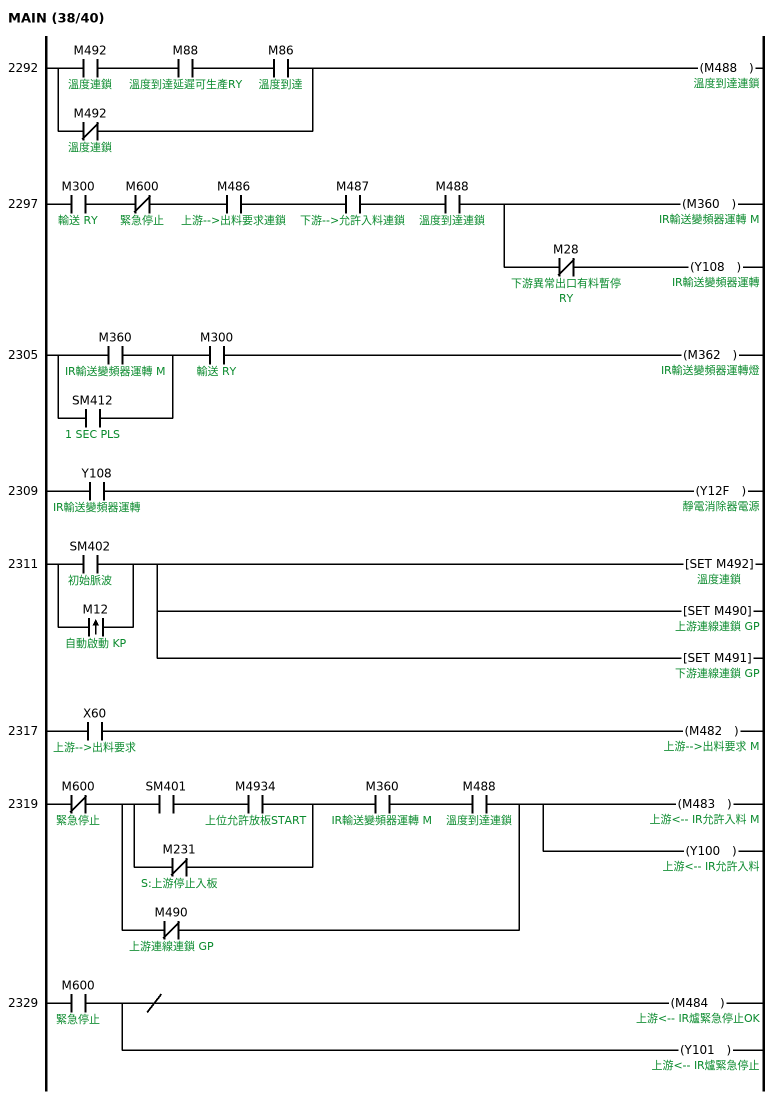
2292  LD      M492  ; 溫度連鎖
      AND     M88  ; 溫度到達延遲可生產RY
      AND     M86  ; 溫度到達
      ORI     M492  ; 溫度連鎖
      OUT     M488  ; 溫度到達連鎖
2297  LD      M300  ; 輸送 RY
      ANI     M600  ; 緊急停止
      AND     M486  ; 上游-->出料要求連鎖
      AND     M487  ; 下游-->允許入料連鎖
      AND     M488  ; 溫度到達連鎖
      OUT     M360  ; IR輸送變頻器運轉 M
      ANI     M28  ; 下游異常出口有料暫停 RY
      OUT     Y108  ; IR輸送變頻器運轉
2305  LD      M360  ; IR輸送變頻器運轉 M
      OR      SM412  ; 1 SEC PLS
      AND     M300  ; 輸送 RY
      OUT     M362  ; IR輸送變頻器運轉燈
2309  LD      Y108  ; IR輸送變頻器運轉
      OUT     Y12F  ; 靜電消除器電源
2311  LD      SM402  ; 初始脈波
      ORP     M12  ; 自動啟動 KP
      SET     M492  ; 溫度連鎖
      SET     M490  ; 上游連線連鎖 GP
      SET     M491  ; 下游連線連鎖 GP
2317  LD      X60  ; 上游-->出料要求
      OUT     M482  ; 上游-->出料要求 M
2319  LDI     M600  ; 緊急停止
      LD      SM401
      AND     M4934  ; 上位允許放板START
      ORI     M231  ; S:上游停止入板
      AND     M360  ; IR輸送變頻器運轉 M
      AND     M488  ; 溫度到達連鎖
      ORI     M490  ; 上游連線連鎖 GP
      ANB
      OUT     M483  ; 上游<-- IR允許入料 M
      OUT     Y100  ; 上游<-- IR允許入料
2329  LD      M600  ; 緊急停止
      MPS
      INV
      OUT     M484  ; 上游<-- IR爐緊急停止OK
      MPP
      OUT     Y101  ; 上游<-- IR爐緊急停止
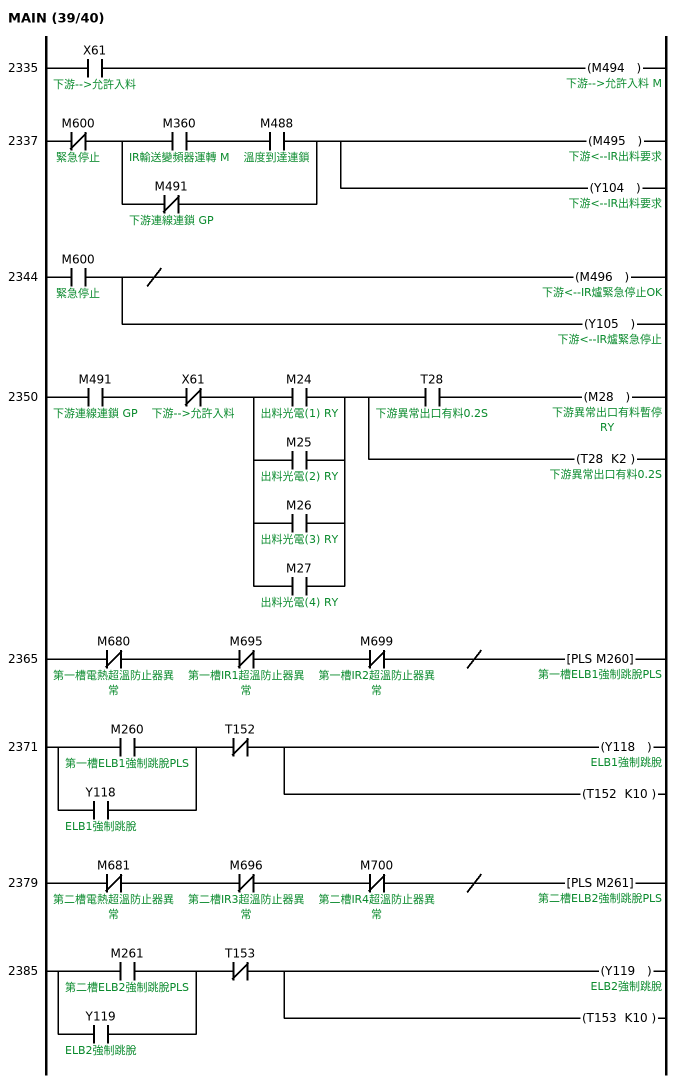
2335  LD      X61  ; 下游-->允許入料
      OUT     M494  ; 下游-->允許入料 M
2337  LDI     M600  ; 緊急停止
      LD      M360  ; IR輸送變頻器運轉 M
      AND     M488  ; 溫度到達連鎖
      ORI     M491  ; 下游連線連鎖 GP
      ANB
      OUT     M495  ; 下游<--IR出料要求
      OUT     Y104  ; 下游<--IR出料要求
2344  LD      M600  ; 緊急停止
      MPS
      INV
      OUT     M496  ; 下游<--IR爐緊急停止OK
      MPP
      OUT     Y105  ; 下游<--IR爐緊急停止
2350  LD      M491  ; 下游連線連鎖 GP
      ANI     X61  ; 下游-->允許入料
      LD      M24  ; 出料光電(1) RY
      OR      M25  ; 出料光電(2) RY
      OR      M26  ; 出料光電(3) RY
      OR      M27  ; 出料光電(4) RY
      ANB
      MPS
      AND     T28  ; 下游異常出口有料0.2S
      OUT     M28  ; 下游異常出口有料暫停 RY
      MPP
      OUT     T28 K2  ; 下游異常出口有料0.2S
2365  LDI     M680  ; 第一槽電熱超溫防止器異常
      ANI     M695  ; 第一槽IR1超溫防止器異常
      ANI     M699  ; 第一槽IR2超溫防止器異常
      INV
      PLS     M260  ; 第一槽ELB1強制跳脫PLS
2371  LD      M260  ; 第一槽ELB1強制跳脫PLS
      OR      Y118  ; ELB1強制跳脫
      ANI     T152
      OUT     Y118  ; ELB1強制跳脫
      OUT     T152 K10
2379  LDI     M681  ; 第二槽電熱超溫防止器異常
      ANI     M696  ; 第二槽IR3超溫防止器異常
      ANI     M700  ; 第二槽IR4超溫防止器異常
      INV
      PLS     M261  ; 第二槽ELB2強制跳脫PLS
2385  LD      M261  ; 第二槽ELB2強制跳脫PLS
      OR      Y119  ; ELB2強制跳脫
      ANI     T153
      OUT     Y119  ; ELB2強制跳脫
      OUT     T153 K10
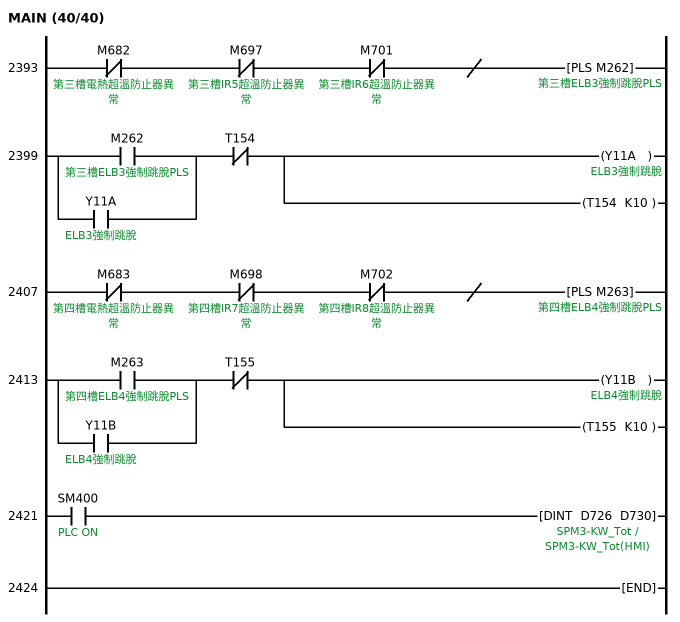
2393  LDI     M682  ; 第三槽電熱超溫防止器異常
      ANI     M697  ; 第三槽IR5超溫防止器異常
      ANI     M701  ; 第三槽IR6超溫防止器異常
      INV
      PLS     M262  ; 第三槽ELB3強制跳脫PLS
2399  LD      M262  ; 第三槽ELB3強制跳脫PLS
      OR      Y11A  ; ELB3強制跳脫
      ANI     T154
      OUT     Y11A  ; ELB3強制跳脫
      OUT     T154 K10
2407  LDI     M683  ; 第四槽電熱超溫防止器異常
      ANI     M698  ; 第四槽IR7超溫防止器異常
      ANI     M702  ; 第四槽IR8超溫防止器異常
      INV
      PLS     M263  ; 第四槽ELB4強制跳脫PLS
2413  LD      M263  ; 第四槽ELB4強制跳脫PLS
      OR      Y11B  ; ELB4強制跳脫
      ANI     T155
      OUT     Y11B  ; ELB4強制跳脫
      OUT     T155 K10
2421  LD      SM400  ; PLC ON
      DINT    D726 D730  ; SPM3-KW_Tot / SPM3-KW_Tot(HMI)
2424  END
END_PROGRAM

PROGRAM SECS
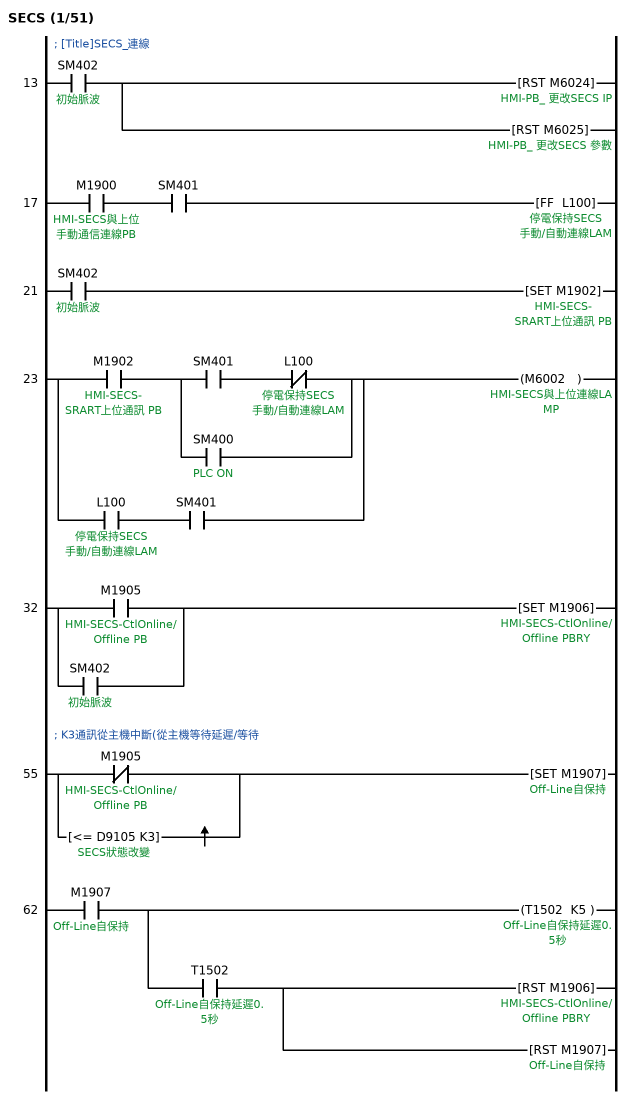
; [Title]SECS_連線
13    LD      SM402  ; 初始脈波
      RST     M6024  ; HMI-PB_ 更改SECS IP
      RST     M6025  ; HMI-PB_ 更改SECS 參數
17    LD      M1900  ; HMI-SECS與上位 手動通信連線PB
      AND     SM401
      FF      L100  ; 停電保持SECS  手動/自動連線LAM
21    LD      SM402  ; 初始脈波
      SET     M1902  ; HMI-SECS-SRART上位通訊 PB
23    LD      M1902  ; HMI-SECS-SRART上位通訊 PB
      LD      SM401
      ANI     L100  ; 停電保持SECS  手動/自動連線LAM
      OR      SM400  ; PLC ON
      ANB
      LD      L100  ; 停電保持SECS  手動/自動連線LAM
      AND     SM401
      ORB
      OUT     M6002  ; HMI-SECS與上位連線LAMP
32    LD      M1905  ; HMI-SECS-CtlOnline/ Offline PB
      OR      SM402  ; 初始脈波
      SET     M1906  ; HMI-SECS-CtlOnline/ Offline PBRY
; K3通訊從主機中斷(從主機等待延遲/等待
55    LDI     M1905  ; HMI-SECS-CtlOnline/ Offline PB
      LD<=    D9105 K3  ; SECS狀態改變
      MEP
      ORB
      SET     M1907  ; Off-Line自保持
62    LD      M1907  ; Off-Line自保持
      OUT     T1502 K5  ; Off-Line自保持延遲0.5秒
      AND     T1502  ; Off-Line自保持延遲0.5秒
      RST     M1906  ; HMI-SECS-CtlOnline/ Offline PBRY
      RST     M1907  ; Off-Line自保持
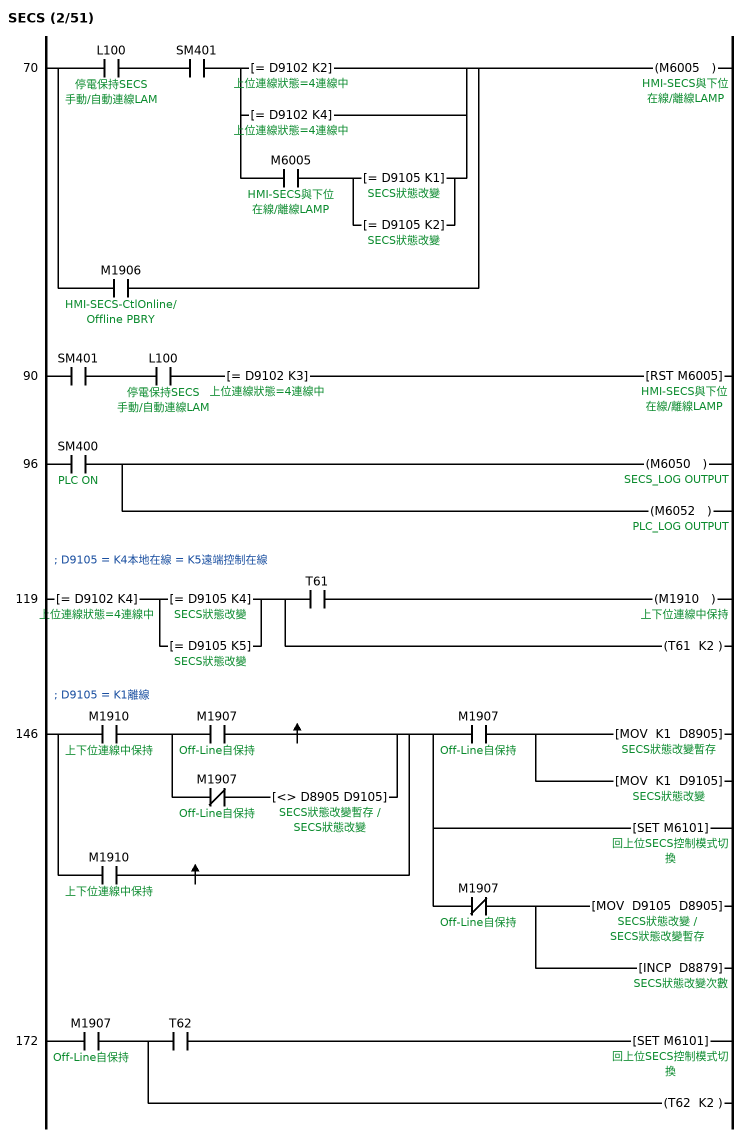
70    LD      L100  ; 停電保持SECS  手動/自動連線LAM
      AND     SM401
      LD=     D9102 K2  ; 上位連線狀態=4連線中
      OR=     D9102 K4  ; 上位連線狀態=4連線中
      LD      M6005  ; HMI-SECS與下位 在線/離線LAMP
      LD=     D9105 K1  ; SECS狀態改變
      OR=     D9105 K2  ; SECS狀態改變
      ANB
      ORB
      ANB
      OR      M1906  ; HMI-SECS-CtlOnline/ Offline PBRY
      OUT     M6005  ; HMI-SECS與下位 在線/離線LAMP
90    LD      SM401
      AND     L100  ; 停電保持SECS  手動/自動連線LAM
      AND=    D9102 K3  ; 上位連線狀態=4連線中
      RST     M6005  ; HMI-SECS與下位 在線/離線LAMP
96    LD      SM400  ; PLC ON
      OUT     M6050  ; SECS_LOG OUTPUT
      OUT     M6052  ; PLC_LOG OUTPUT
; D9105 = K4本地在線 = K5遠端控制在線
119   LD=     D9102 K4  ; 上位連線狀態=4連線中
      LD=     D9105 K4  ; SECS狀態改變
      OR=     D9105 K5  ; SECS狀態改變
      ANB
      MPS
      AND     T61
      OUT     M1910  ; 上下位連線中保持
      MPP
      OUT     T61 K2
; D9105 = K1離線
146   LD      M1910  ; 上下位連線中保持
      LD      M1907  ; Off-Line自保持
      MEP
      LDI     M1907  ; Off-Line自保持
      AND<>   D8905 D9105  ; SECS狀態改變暫存 / SECS狀態改變
      ORB
      ANB
      LD      M1910  ; 上下位連線中保持
      MEP
      ORB
      MPS
      AND     M1907  ; Off-Line自保持
      MOV     K1 D8905
      MOV     K1 D9105
      MPP
      SET     M6101  ; 回上位SECS控制模式切換
      ANI     M1907  ; Off-Line自保持
      MOV     D9105 D8905
      INCP    D8879  ; SECS狀態改變次數
172   LD      M1907  ; Off-Line自保持
      MPS
      AND     T62
      SET     M6101  ; 回上位SECS控制模式切換
      MPP
      OUT     T62 K2
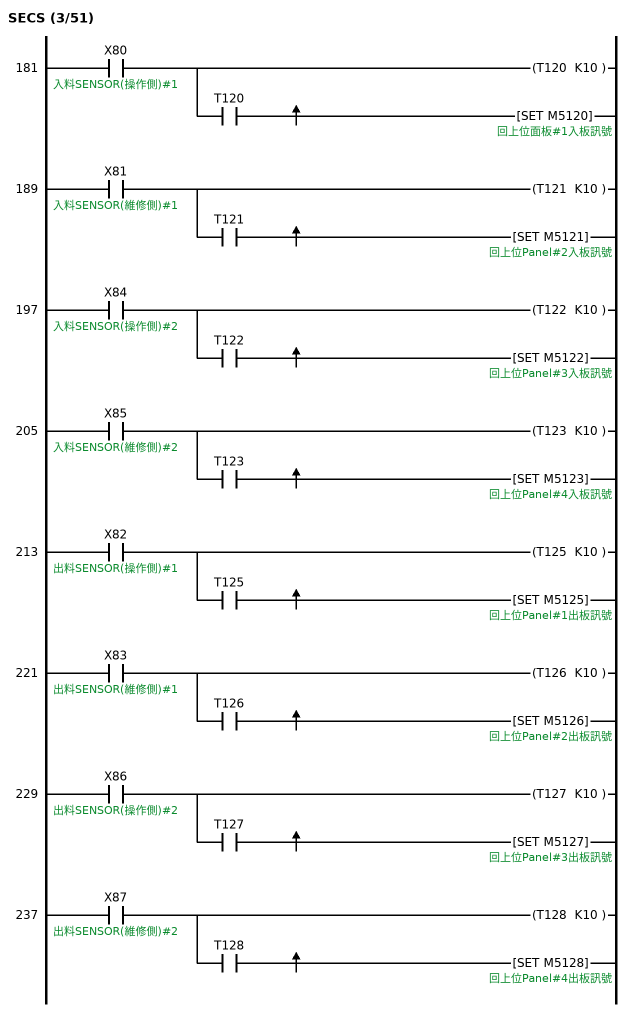
181   LD      X80  ; 入料SENSOR(操作側)#1
      OUT     T120 K10
      AND     T120
      MEP
      SET     M5120  ; 回上位面板#1入板訊號
189   LD      X81  ; 入料SENSOR(維修側)#1
      OUT     T121 K10
      AND     T121
      MEP
      SET     M5121  ; 回上位Panel#2入板訊號
197   LD      X84  ; 入料SENSOR(操作側)#2
      OUT     T122 K10
      AND     T122
      MEP
      SET     M5122  ; 回上位Panel#3入板訊號
205   LD      X85  ; 入料SENSOR(維修側)#2
      OUT     T123 K10
      AND     T123
      MEP
      SET     M5123  ; 回上位Panel#4入板訊號
213   LD      X82  ; 出料SENSOR(操作側)#1
      OUT     T125 K10
      AND     T125
      MEP
      SET     M5125  ; 回上位Panel#1出板訊號
221   LD      X83  ; 出料SENSOR(維修側)#1
      OUT     T126 K10
      AND     T126
      MEP
      SET     M5126  ; 回上位Panel#2出板訊號
229   LD      X86  ; 出料SENSOR(操作側)#2
      OUT     T127 K10
      AND     T127
      MEP
      SET     M5127  ; 回上位Panel#3出板訊號
237   LD      X87  ; 出料SENSOR(維修側)#2
      OUT     T128 K10
      AND     T128
      MEP
      SET     M5128  ; 回上位Panel#4出板訊號
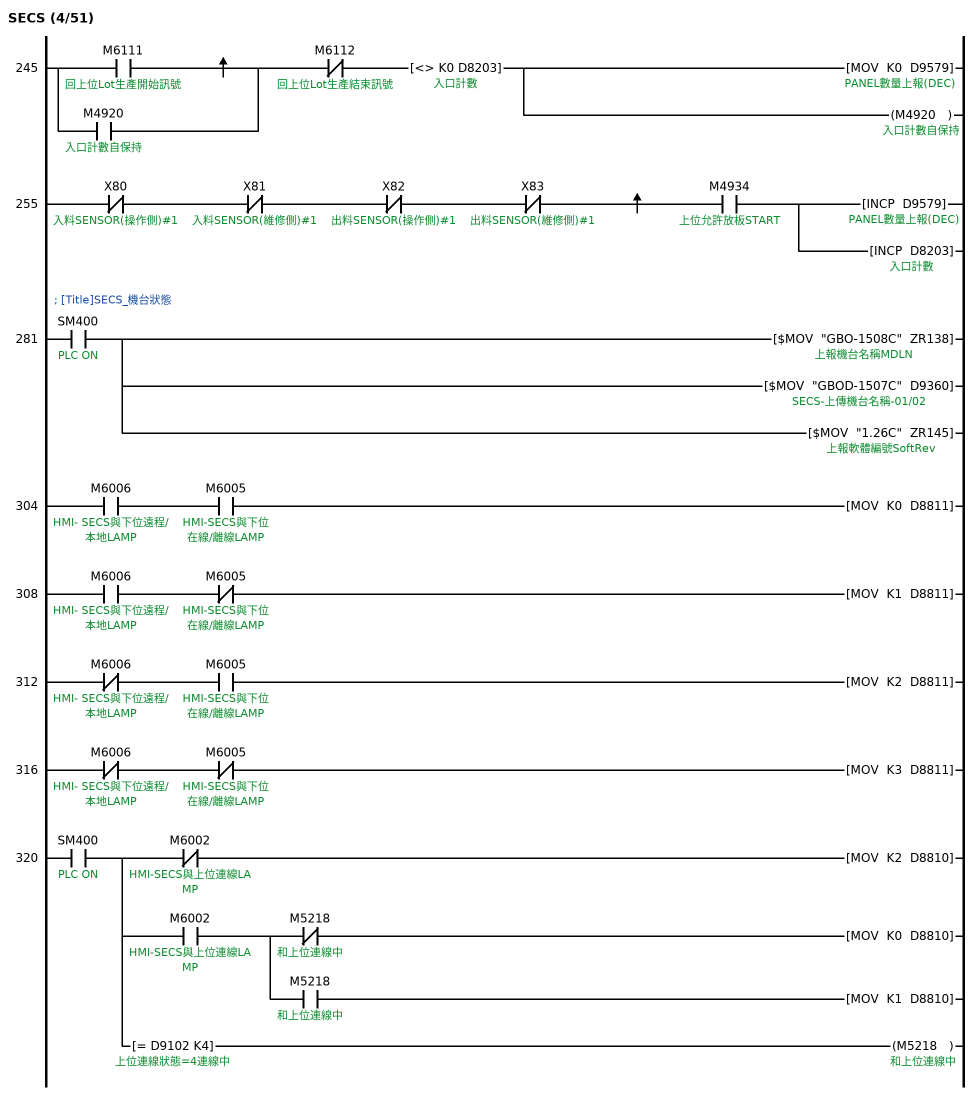
245   LD      M6111  ; 回上位Lot生產開始訊號
      MEP
      OR      M4920  ; 入口計數自保持
      ANI     M6112  ; 回上位Lot生產結束訊號
      AND<>   K0 D8203  ; 入口計數
      MOV     K0 D9579  ; PANEL數量上報(DEC)
      OUT     M4920  ; 入口計數自保持
255   LDI     X80  ; 入料SENSOR(操作側)#1
      ANI     X81  ; 入料SENSOR(維修側)#1
      ANI     X82  ; 出料SENSOR(操作側)#1
      ANI     X83  ; 出料SENSOR(維修側)#1
      MEP
      AND     M4934  ; 上位允許放板START
      INCP    D9579
      INCP    D8203
; [Title]SECS_機台狀態
281   LD      SM400  ; PLC ON
      $MOV    "GBO-1508C" ZR138  ; 上報機台名稱MDLN
      $MOV    "GBOD-1507C" D9360  ; SECS-上傳機台名稱-01/02
      $MOV    "1.26C" ZR145  ; 上報軟體編號SoftRev
304   LD      M6006  ; HMI- SECS與下位遠程/本地LAMP
      AND     M6005  ; HMI-SECS與下位 在線/離線LAMP
      MOV     K0 D8811
308   LD      M6006  ; HMI- SECS與下位遠程/本地LAMP
      ANI     M6005  ; HMI-SECS與下位 在線/離線LAMP
      MOV     K1 D8811
312   LDI     M6006  ; HMI- SECS與下位遠程/本地LAMP
      AND     M6005  ; HMI-SECS與下位 在線/離線LAMP
      MOV     K2 D8811
316   LDI     M6006  ; HMI- SECS與下位遠程/本地LAMP
      ANI     M6005  ; HMI-SECS與下位 在線/離線LAMP
      MOV     K3 D8811
320   LD      SM400  ; PLC ON
      MPS
      ANI     M6002  ; HMI-SECS與上位連線LAMP
      MOV     K2 D8810
      MRD
      AND     M6002  ; HMI-SECS與上位連線LAMP
      MPS
      ANI     M5218  ; 和上位連線中
      MOV     K0 D8810
      MPP
      AND     M5218  ; 和上位連線中
      MOV     K1 D8810
      MPP
      AND=    D9102 K4  ; 上位連線狀態=4連線中
      OUT     M5218  ; 和上位連線中
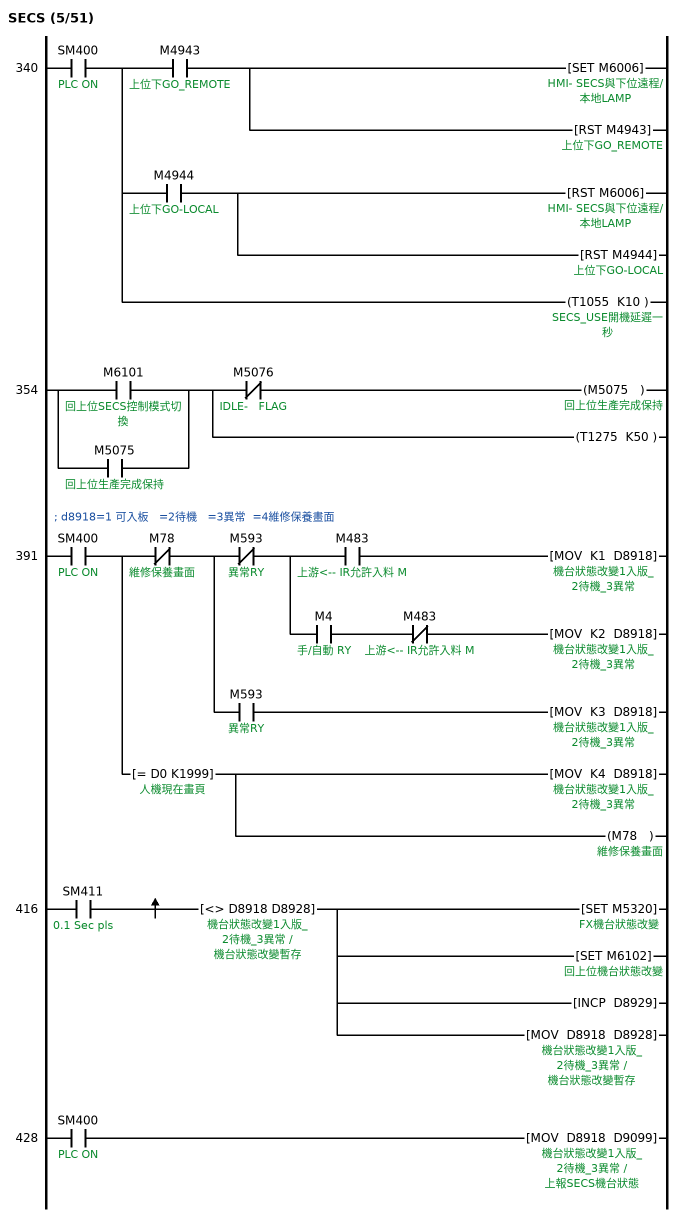
340   LD      SM400  ; PLC ON
      MPS
      AND     M4943  ; 上位下GO_REMOTE
      SET     M6006  ; HMI- SECS與下位遠程/本地LAMP
      RST     M4943  ; 上位下GO_REMOTE
      MRD
      AND     M4944  ; 上位下GO-LOCAL
      RST     M6006  ; HMI- SECS與下位遠程/本地LAMP
      RST     M4944  ; 上位下GO-LOCAL
      MPP
      OUT     T1055 K10  ; SECS_USE開機延遲一秒
354   LD      M6101  ; 回上位SECS控制模式切換
      OR      M5075  ; 回上位生產完成保持
      MPS
      ANI     M5076  ; IDLE-   FLAG
      OUT     M5075  ; 回上位生產完成保持
      MPP
      OUT     T1275 K50
; d8918=1 可入板   =2待機   =3異常  =4維修保養畫面
391   LD      SM400  ; PLC ON
      MPS
      ANI     M78  ; 維修保養畫面
      MPS
      ANI     M593  ; 異常RY
      MPS
      AND     M483  ; 上游<-- IR允許入料 M
      MOV     K1 D8918  ; 機台狀態改變1入版_2待機_3異常
      MPP
      AND     M4  ; 手/自動 RY
      ANI     M483  ; 上游<-- IR允許入料 M
      MOV     K2 D8918
      MPP
      AND     M593  ; 異常RY
      MOV     K3 D8918
      MPP
      AND=    D0 K1999  ; 人機現在畫頁
      MOV     K4 D8918
      OUT     M78  ; 維修保養畫面
416   LD      SM411  ; 0.1 Sec pls
      MEP
      AND<>   D8918 D8928  ; 機台狀態改變1入版_2待機_3異常 / 機台狀態改變暫存
      SET     M5320  ; FX機台狀態改變
      SET     M6102  ; 回上位機台狀態改變
      INCP    D8929
      MOV     D8918 D8928
428   LD      SM400  ; PLC ON
      MOV     D8918 D9099  ; 上報SECS機台狀態
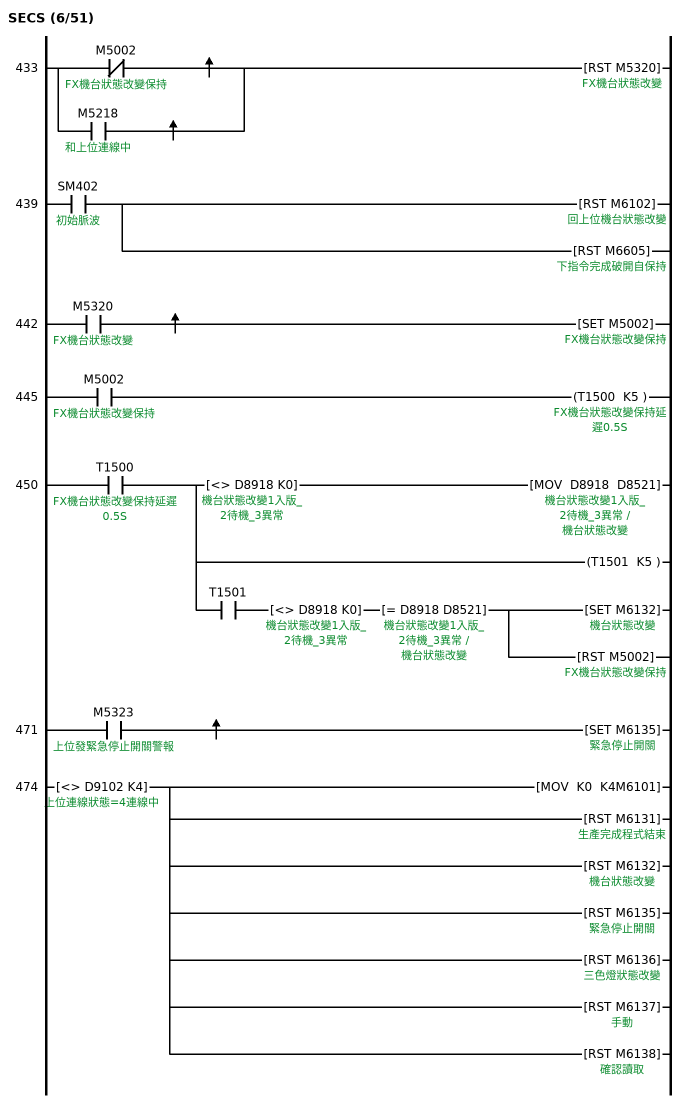
433   LDI     M5002  ; FX機台狀態改變保持
      MEP
      LD      M5218  ; 和上位連線中
      MEP
      ORB
      RST     M5320  ; FX機台狀態改變
439   LD      SM402  ; 初始脈波
      RST     M6102  ; 回上位機台狀態改變
      RST     M6605  ; 下指令完成破開自保持
442   LD      M5320  ; FX機台狀態改變
      MEP
      SET     M5002  ; FX機台狀態改變保持
445   LD      M5002  ; FX機台狀態改變保持
      OUT     T1500 K5  ; FX機台狀態改變保持延遲0.5S
450   LD      T1500  ; FX機台狀態改變保持延遲0.5S
      MPS
      AND<>   D8918 K0  ; 機台狀態改變1入版_2待機_3異常
      MOV     D8918 D8521  ; 機台狀態改變
      MPP
      OUT     T1501 K5
      AND     T1501
      AND<>   D8918 K0  ; 機台狀態改變1入版_2待機_3異常
      AND=    D8918 D8521  ; 機台狀態改變1入版_2待機_3異常 / 機台狀態改變
      SET     M6132  ; 機台狀態改變
      RST     M5002  ; FX機台狀態改變保持
471   LD      M5323  ; 上位發緊急停止開關警報
      MEP
      SET     M6135  ; 緊急停止開關
474   LD<>    D9102 K4  ; 上位連線狀態=4連線中
      MOV     K0 K4M6101
      RST     M6131  ; 生產完成程式結束
      RST     M6132  ; 機台狀態改變
      RST     M6135  ; 緊急停止開關
      RST     M6136  ; 三色燈狀態改變
      RST     M6137  ; 手動
      RST     M6138  ; 確認讀取
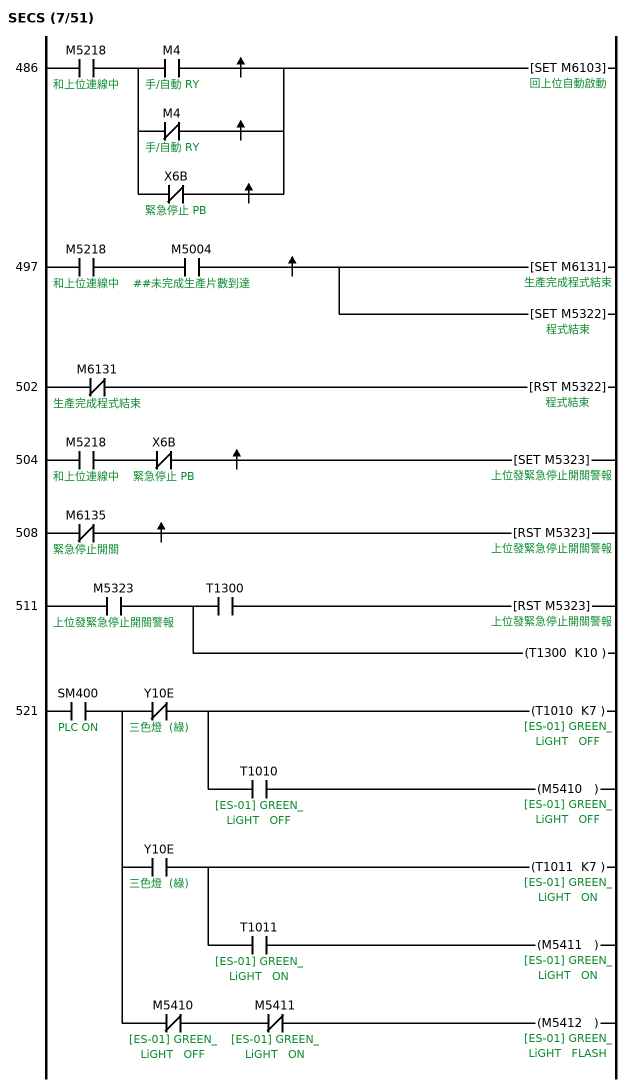
486   LD      M5218  ; 和上位連線中
      LD      M4  ; 手/自動 RY
      MEP
      LDI     M4  ; 手/自動 RY
      MEP
      ORB
      LDI     X6B  ; 緊急停止 PB
      MEP
      ORB
      ANB
      SET     M6103  ; 回上位自動啟動
497   LD      M5218  ; 和上位連線中
      AND     M5004  ; ##未完成生產片數到達
      MEP
      SET     M6131  ; 生產完成程式結束
      SET     M5322  ; 程式結束
502   LDI     M6131  ; 生產完成程式結束
      RST     M5322  ; 程式結束
504   LD      M5218  ; 和上位連線中
      ANI     X6B  ; 緊急停止 PB
      MEP
      SET     M5323  ; 上位發緊急停止開關警報
508   LDI     M6135  ; 緊急停止開關
      MEP
      RST     M5323  ; 上位發緊急停止開關警報
511   LD      M5323  ; 上位發緊急停止開關警報
      MPS
      AND     T1300
      RST     M5323  ; 上位發緊急停止開關警報
      MPP
      OUT     T1300 K10
521   LD      SM400  ; PLC ON
      MPS
      ANI     Y10E  ; 三色燈  (綠)
      OUT     T1010 K7  ; [ES-01] GREEN_  LiGHT   OFF
      AND     T1010  ; [ES-01] GREEN_  LiGHT   OFF
      OUT     M5410  ; [ES-01] GREEN_  LiGHT   OFF
      MRD
      AND     Y10E  ; 三色燈  (綠)
      OUT     T1011 K7  ; [ES-01] GREEN_  LiGHT   ON
      AND     T1011  ; [ES-01] GREEN_  LiGHT   ON
      OUT     M5411  ; [ES-01] GREEN_  LiGHT   ON
      MPP
      ANI     M5410  ; [ES-01] GREEN_  LiGHT   OFF
      ANI     M5411  ; [ES-01] GREEN_  LiGHT   ON
      OUT     M5412  ; [ES-01] GREEN_  LiGHT   FLASH
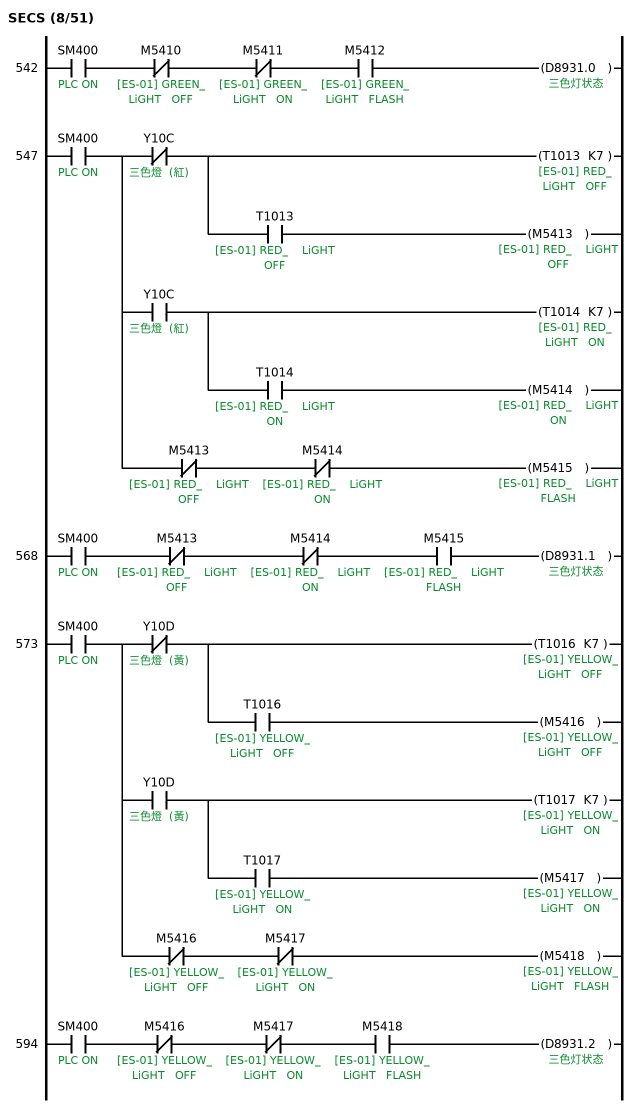
542   LD      SM400  ; PLC ON
      ANI     M5410  ; [ES-01] GREEN_  LiGHT   OFF
      ANI     M5411  ; [ES-01] GREEN_  LiGHT   ON
      AND     M5412  ; [ES-01] GREEN_  LiGHT   FLASH
      OUT     D8931.0  ; 三色灯状态
547   LD      SM400  ; PLC ON
      MPS
      ANI     Y10C  ; 三色燈  (紅)
      OUT     T1013 K7  ; [ES-01] RED_    LiGHT   OFF
      AND     T1013  ; [ES-01] RED_    LiGHT   OFF
      OUT     M5413  ; [ES-01] RED_    LiGHT   OFF
      MRD
      AND     Y10C  ; 三色燈  (紅)
      OUT     T1014 K7  ; [ES-01] RED_    LiGHT   ON
      AND     T1014  ; [ES-01] RED_    LiGHT   ON
      OUT     M5414  ; [ES-01] RED_    LiGHT   ON
      MPP
      ANI     M5413  ; [ES-01] RED_    LiGHT   OFF
      ANI     M5414  ; [ES-01] RED_    LiGHT   ON
      OUT     M5415  ; [ES-01] RED_    LiGHT   FLASH
568   LD      SM400  ; PLC ON
      ANI     M5413  ; [ES-01] RED_    LiGHT   OFF
      ANI     M5414  ; [ES-01] RED_    LiGHT   ON
      AND     M5415  ; [ES-01] RED_    LiGHT   FLASH
      OUT     D8931.1  ; 三色灯状态
573   LD      SM400  ; PLC ON
      MPS
      ANI     Y10D  ; 三色燈  (黃)
      OUT     T1016 K7  ; [ES-01] YELLOW_ LiGHT   OFF
      AND     T1016  ; [ES-01] YELLOW_ LiGHT   OFF
      OUT     M5416  ; [ES-01] YELLOW_ LiGHT   OFF
      MRD
      AND     Y10D  ; 三色燈  (黃)
      OUT     T1017 K7  ; [ES-01] YELLOW_ LiGHT   ON
      AND     T1017  ; [ES-01] YELLOW_ LiGHT   ON
      OUT     M5417  ; [ES-01] YELLOW_ LiGHT   ON
      MPP
      ANI     M5416  ; [ES-01] YELLOW_ LiGHT   OFF
      ANI     M5417  ; [ES-01] YELLOW_ LiGHT   ON
      OUT     M5418  ; [ES-01] YELLOW_ LiGHT   FLASH
594   LD      SM400  ; PLC ON
      ANI     M5416  ; [ES-01] YELLOW_ LiGHT   OFF
      ANI     M5417  ; [ES-01] YELLOW_ LiGHT   ON
      AND     M5418  ; [ES-01] YELLOW_ LiGHT   FLASH
      OUT     D8931.2  ; 三色灯状态
